// TwinCAT 3 PLC project plc_kfe_rix_vac
// Title: plc-kfe-rix-vac
// Company: SLAC
// ProjectVersion: 0.0.0
// ProgramVersion: 3.1.4023.0
// libraries:
//   LCLS General, * (SLAC)
//   LCLS Vacuum, * (SLAC - LCLS)
//   LCLSVacuumSerialDriverLib, * (SLAC)
//   PMPS, * (SLAC - LCLS)
//   Tc2_DataExchange, * (Beckhoff Automation GmbH)
//   Tc2_SerialCom, * (Beckhoff Automation GmbH)
//   Tc2_Standard, * (Beckhoff Automation GmbH)
//   Tc2_System, * (Beckhoff Automation GmbH)
//   Tc2_TcpIp, * (Beckhoff Automation GmbH)
//   Tc2_Utilities, * (Beckhoff Automation GmbH)
//   Tc3_Module, * (Beckhoff Automation GmbH)
// project tree:
//   / CheckBounds.TcPOU (not stored), CheckDivDInt.TcPOU (not stored), CheckDivLInt.TcPOU (not stored), CheckDivLReal.TcPOU (not stored), CheckDivReal.TcPOU (not stored), CheckLRangeSigned.TcPOU (not stored), CheckLRangeUnsigned.TcPOU (not stored), CheckPointer.TcPOU (not stored), CheckRangeSigned.TcPOU (not stored), CheckRangeUnsigned.TcPOU (not stored), FSTask.TcTTO (not stored), PlcTask.TcTTO (not stored), Serial_COM.TcTTO (not stored)
//   DUTs/ ST_EXT_ILK.TcDUT (not stored)
//   GVLs/ GVL_RIX_INTF.TcGVL (not stored), GVL_KFE_RIX_VAC.TcGVL, GVL_RIX_VAC_FSV_PMPS.TcGVL (not stored), GVL_RIX_VAC_FS_DEVICES.TcGVL (not stored), GVL_Serial_Com.TcGVL, GVL_Variables.TcGVL
//   POUs/ FB_PRO_ADS.TcPOU (not stored), MAIN.TcPOU (not stored), FB_EXT_ILK.TcPOU (not stored), PRG_COM.TcPOU, PRG_RIX_INTF.TcPOU (not stored), PRG_KFE_RIX_VAC.TcPOU, PRG_KFE_RIX_VAC_FS.TcPOU (not stored), PRG_Roughing.TcPOU (not stored)
// real-time tasks:
//   TASK PlcTask: cycle T#10ms, priority 20, ADS port 350
//   TASK FSTask: cycle T#1ms, priority 19, ADS port 352
//   TASK Serial_COM: cycle T#10ms, priority 25, ADS port 351
// I/O:
//   DEVICE Device 1 (EtherCAT)
//   DEVICE Device 5 (EtherCAT)
// variable links:
//   plc_kfe_rix_vac Instance <-> Device 1 (EtherCAT)/B950_100H1_WALL (EK1100)/Term 118 (EL2624)
//     PlcTask Outputs/GVL_KFE_RIX_VAC.fb_SL1K2_EXIT_GCC_1.q_xHV_DIS <-> Channel 1/Output
//   plc_kfe_rix_vac Instance <-> Device 1 (EtherCAT)/B950_100H1_WALL (EK1100)/Term 119 (EL3174)
//     PlcTask Inputs/GVL_KFE_RIX_VAC.fb_SL1K2_EXIT_GCC_1.i_iPRESS_R <-> AI Standard Channel 1/Value
//     PlcTask Inputs/GVL_KFE_RIX_VAC.fb_SL1K2_EXIT_GPI_1.i_iPRESS_R <-> AI Standard Channel 2/Value
//   plc_kfe_rix_vac Instance <-> Device 1 (EtherCAT)/B950_100H1_WALL (EK1100)/Term 120 (EL1004)
//     PlcTask Inputs/GVL_KFE_RIX_VAC.fb_SL1K2_EXIT_VGC_1.i_xClsLS <-> Channel 2/Input
//     PlcTask Inputs/GVL_KFE_RIX_VAC.fb_SL1K2_EXIT_VGC_1.i_xOpnLS <-> Channel 1/Input
//   plc_kfe_rix_vac Instance <-> Device 1 (EtherCAT)/B950_100H1_WALL (EK1100)/Term 121 (EL2004)
//     PlcTask Outputs/GVL_KFE_RIX_VAC.fb_SL1K2_EXIT_VGC_1.q_xOPN_DO <-> Channel 1/Output
//   plc_kfe_rix_vac Instance <-> Device 1 (EtherCAT)/B950_100H1_WALL (EK1100)/Term 123 (EL1124)
//     PlcTask Inputs/GVL_KFE_RIX_VAC.fb_SL1K2_EXIT_GCC_1.i_xDisc_Active <-> Channel 2/Input
//     PlcTask Inputs/GVL_KFE_RIX_VAC.fb_SL1K2_EXIT_GCC_1.i_xHV_ON <-> Channel 1/Input
//   plc_kfe_rix_vac Instance <-> Device 1 (EtherCAT)/Term 1 (EK1200)/PMPS_FFO (EL2202)
//     FSTask Outputs/GVL_RIX_VAC_FSV_PMPS.g_FastFaultOutput2.q_xFastFaultOut <-> Channel 2/Output
//     PlcTask Outputs/GVL_Variables.g_FastFaultOutput1.q_xFastFaultOut <-> Channel 1/Output
//   plc_kfe_rix_vac Instance <-> Device 1 (EtherCAT)/Term 1 (EK1200)/PMPS_PRE
//     PlcTask Inputs/MAIN.fbArbiterIO.i_stCurrentBP <-> IO Inputs/CurrentBP
//     PlcTask Inputs/MAIN.fbArbiterIO.xTxPDO_state <-> SYNC Inputs/TxPDO state
//     PlcTask Inputs/MAIN.fbArbiterIO.xTxPDO_toggle <-> SYNC Inputs/TxPDO toggle
//     PlcTask Outputs/MAIN.fbArbiterIO.q_stRequestedBP <-> IO Outputs/RequestedBP
//   plc_kfe_rix_vac Instance <-> Device 1 (EtherCAT)/Term 1 (EK1200)/Term 11 (EL2794)
//     PlcTask Outputs/GVL_KFE_RIX_VAC.fb_RIX_ILK.q_xILK_OK_DO <-> Channel 1/Output
//   plc_kfe_rix_vac Instance <-> Device 1 (EtherCAT)/Term 1 (EK1200)/Term 3 (EL2794)
//     PlcTask Outputs/GVL_KFE_RIX_VAC.fb_MR1K2_SWITCH_PIP_1.q_xHVEna_DO <-> Channel 3/Output
//     PlcTask Outputs/GVL_KFE_RIX_VAC.fb_PC1K1_ZOS_PIP_1.q_xHVEna_DO <-> Channel 2/Output
//     PlcTask Outputs/GVL_KFE_RIX_VAC.fb_TV1K1_PLEG_PIP_1.q_xHVEna_DO <-> Channel 4/Output
//   plc_kfe_rix_vac Instance <-> Device 1 (EtherCAT)/Term 1 (EK1200)/Term 32 (EK1122)/B940-008-K0S15-PNL-03 EK1100/Term 13 (EL2624)
//     PlcTask Outputs/GVL_KFE_RIX_VAC.fb_MR1K2_SWITCH_GCC_1.q_xHV_DIS <-> Channel 3/Output
//     PlcTask Outputs/GVL_KFE_RIX_VAC.fb_PC1K1_ZOS_GCC_1.q_xHV_DIS <-> Channel 1/Output
//     PlcTask Outputs/GVL_KFE_RIX_VAC.fb_TV1K1_PLEG_GCC_1.q_xHV_DIS <-> Channel 2/Output
//   plc_kfe_rix_vac Instance <-> Device 1 (EtherCAT)/Term 1 (EK1200)/Term 32 (EK1122)/B940-008-K0S15-PNL-03 EK1100/Term 14 (EL1004)
//     PlcTask Inputs/GVL_KFE_RIX_VAC.fb_MR1K2_SWITCH_VGC_1.i_xClsLS <-> Channel 2/Input
//     PlcTask Inputs/GVL_KFE_RIX_VAC.fb_MR1K2_SWITCH_VGC_2.i_xClsLS <-> Channel 4/Input
//     PlcTask Inputs/GVL_KFE_RIX_VAC.fb_MR1K2_SWITCH_VGC_1.i_xOpnLS <-> Channel 1/Input
//     PlcTask Inputs/GVL_KFE_RIX_VAC.fb_MR1K2_SWITCH_VGC_2.i_xOpnLS <-> Channel 3/Input
//   plc_kfe_rix_vac Instance <-> Device 1 (EtherCAT)/Term 1 (EK1200)/Term 32 (EK1122)/B940-008-K0S15-PNL-03 EK1100/Term 15 (EL2004)
//     PlcTask Outputs/GVL_KFE_RIX_VAC.fb_MR1K2_SWITCH_VGC_1.q_xOPN_DO <-> Channel 1/Output
//     PlcTask Outputs/GVL_KFE_RIX_VAC.fb_MR1K2_SWITCH_VGC_2.q_xOPN_DO <-> Channel 2/Output
//   plc_kfe_rix_vac Instance <-> Device 1 (EtherCAT)/Term 1 (EK1200)/Term 32 (EK1122)/B940-008-K0S15-PNL-03 EK1100/Term 16 (EL3174-0002)
//     PlcTask Inputs/GVL_KFE_RIX_VAC.fb_MR1K2_SWITCH_GCC_1.i_iPRESS_R <-> AI Standard Channel 2/Value
//     PlcTask Inputs/GVL_KFE_RIX_VAC.fb_PC1K1_ZOS_GCC_1.i_iPRESS_R <-> AI Standard Channel 1/Value
//     PlcTask Inputs/GVL_KFE_RIX_VAC.fb_PC1K1_ZOS_GPI_1.i_iPRESS_R <-> AI Standard Channel 4/Value
//     PlcTask Inputs/GVL_KFE_RIX_VAC.fb_TV1K1_PLEG_GCC_1.i_iPRESS_R <-> AI Standard Channel 3/Value
//   plc_kfe_rix_vac Instance <-> Device 1 (EtherCAT)/Term 1 (EK1200)/Term 32 (EK1122)/B940-008-K0S15-PNL-03 EK1100/Term 17 (EL3174-0002)
//     PlcTask Inputs/GVL_KFE_RIX_VAC.fb_MR1K2_SWITCH_GPI_1.i_iPRESS_R <-> AI Standard Channel 1/Value
//     PlcTask Inputs/GVL_KFE_RIX_VAC.fb_TV1K1_PLEG_GPI_1.i_iPRESS_R <-> AI Standard Channel 2/Value
//   plc_kfe_rix_vac Instance <-> Device 1 (EtherCAT)/Term 1 (EK1200)/Term 32 (EK1122)/B940-008-K0S15-PNL-03 EK1100/Term 19 (EL1124)
//     PlcTask Inputs/GVL_KFE_RIX_VAC.fb_MR1K2_SWITCH_GCC_1.i_xDisc_Active <-> Channel 4/Input
//     PlcTask Inputs/GVL_KFE_RIX_VAC.fb_MR1K2_SWITCH_GCC_1.i_xHV_ON <-> Channel 3/Input
//     PlcTask Inputs/GVL_KFE_RIX_VAC.fb_PC1K1_ZOS_GCC_1.i_xDisc_Active <-> Channel 2/Input
//     PlcTask Inputs/GVL_KFE_RIX_VAC.fb_PC1K1_ZOS_GCC_1.i_xHV_ON <-> Channel 1/Input
//   plc_kfe_rix_vac Instance <-> Device 1 (EtherCAT)/Term 1 (EK1200)/Term 32 (EK1122)/B940-008-K0S15-PNL-03 EK1100/Term 20 (EL1124)
//     PlcTask Inputs/GVL_KFE_RIX_VAC.fb_TV1K1_PLEG_GCC_1.i_xDisc_Active <-> Channel 2/Input
//     PlcTask Inputs/GVL_KFE_RIX_VAC.fb_TV1K1_PLEG_GCC_1.i_xHV_ON <-> Channel 1/Input
//   plc_kfe_rix_vac Instance <-> Device 1 (EtherCAT)/Term 1 (EK1200)/Term 32 (EK1122)/B940-008-K0S15-PNL-03 FS/Term 34 (EL2202)
//     FSTask Outputs/GVL_RIX_VAC_FS_DEVICES.fb_TV1K2_VFS_1.q_xClose_A <-> Channel 1/Output
//     FSTask Outputs/GVL_RIX_VAC_FS_DEVICES.fb_TV1K2_VFS_1.q_xClose_B <-> Channel 2/Output
//   plc_kfe_rix_vac Instance <-> Device 1 (EtherCAT)/Term 1 (EK1200)/Term 32 (EK1122)/B940-008-K0S15-PNL-03 FS/Term 35 (EL2202)
//     FSTask Outputs/GVL_RIX_VAC_FS_DEVICES.fb_TV1K2_VFS_1.q_xClose_C <-> Channel 1/Output
//     FSTask Outputs/GVL_RIX_VAC_FS_DEVICES.fb_TV1K2_VFS_1.q_xOPN_DO <-> Channel 2/Output
//   plc_kfe_rix_vac Instance <-> Device 1 (EtherCAT)/Term 1 (EK1200)/Term 32 (EK1122)/B940-008-K0S15-PNL-03 FS/Term 36 (EL1004)
//     FSTask Inputs/GVL_RIX_VAC_FS_DEVICES.fb_TV1K2_VFS_1.i_xClsLS <-> Channel 1/Input
//     FSTask Inputs/GVL_RIX_VAC_FS_DEVICES.fb_TV1K2_VFS_1.i_xOpnLS <-> Channel 2/Input
//   plc_kfe_rix_vac Instance <-> Device 1 (EtherCAT)/Term 1 (EK1200)/Term 4 (EL3064)
//     PlcTask Inputs/GVL_KFE_RIX_VAC.fb_MR1K2_SWITCH_PIP_1.i_iPRESS <-> AI Standard Channel 3/Value
//     PlcTask Inputs/GVL_KFE_RIX_VAC.fb_PC1K1_ZOS_PIP_1.i_iPRESS <-> AI Standard Channel 2/Value
//     PlcTask Inputs/GVL_KFE_RIX_VAC.fb_TV1K1_PLEG_PIP_1.i_iPRESS <-> AI Standard Channel 4/Value
//   plc_kfe_rix_vac Instance <-> Device 1 (EtherCAT)/Term 1 (EK1200)/Term 45 (EK1521-0010)/Term 47 (EK1501-0010)/B950_233_R02 (E2) (EL2794)
//     PlcTask Outputs/GVL_KFE_RIX_VAC.fb_MR2K2_FLAT_PIP_1.q_xHVEna_DO <-> Channel 2/GVL_KFE_RIX_VAC.fb_MR2K2_FLAT_PIP_1.q_xHVEna_DO
//     PlcTask Outputs/GVL_KFE_RIX_VAC.fb_MR3K2_KBH_PIP_1.q_xHVEna_DO <-> Channel 3/GVL_KFE_RIX_VAC.fb_MR3K2_KBH_PIP_1.q_xHVEna_DO
//     PlcTask Outputs/GVL_KFE_RIX_VAC.fb_MR4K2_KBV_PIP_1.q_xHVEna_DO <-> Channel 4/GVL_KFE_RIX_VAC.fb_MR4K2_KBV_PIP_1.q_xHVEna_DO
//     PlcTask Outputs/GVL_KFE_RIX_VAC.fb_ST1K2_PPS_PIP_1.q_xHVEna_DO <-> Channel 1/GVL_KFE_RIX_VAC.fb_ST1K2_PPS_PIP_1.q_xHVEna_DO
//   plc_kfe_rix_vac Instance <-> Device 1 (EtherCAT)/Term 1 (EK1200)/Term 45 (EK1521-0010)/Term 47 (EK1501-0010)/B950_233_R02 (E3) (EL3064)
//     PlcTask Inputs/GVL_KFE_RIX_VAC.fb_MR2K2_FLAT_PIP_1.i_iPRESS <-> AI Standard Channel 2/GVL_KFE_RIX_VAC.fb_MR2K2_FLAT_PIP_1.i_iPRESS
//     PlcTask Inputs/GVL_KFE_RIX_VAC.fb_MR3K2_KBH_PIP_1.i_iPRESS <-> AI Standard Channel 3/GVL_KFE_RIX_VAC.fb_MR3K2_KBH_PIP_1.i_iPRESS
//     PlcTask Inputs/GVL_KFE_RIX_VAC.fb_MR4K2_KBV_PIP_1.i_iPRESS <-> AI Standard Channel 4/GVL_KFE_RIX_VAC.fb_MR4K2_KBV_PIP_1.i_iPRESS
//     PlcTask Inputs/GVL_KFE_RIX_VAC.fb_ST1K2_PPS_PIP_1.i_iPRESS <-> AI Standard Channel 1/GVL_KFE_RIX_VAC.fb_ST1K2_PPS_PIP_1.i_iPRESS
//   plc_kfe_rix_vac Instance <-> Device 1 (EtherCAT)/Term 1 (EK1200)/Term 45 (EK1521-0010)/Term 47 (EK1501-0010)/B950_233_R02 (E4) (EL1004)
//     PlcTask Inputs/GVL_KFE_RIX_VAC.fb_MR2K2_FLAT_PIP_1.i_xSP_DI <-> Channel 2/GVL_KFE_RIX_VAC.fb_MR2K2_FLAT_PIP_1.i_xSP_DI
//     PlcTask Inputs/GVL_KFE_RIX_VAC.fb_MR3K2_KBH_PIP_1.i_xSP_DI <-> Channel 3/GVL_KFE_RIX_VAC.fb_MR3K2_KBH_PIP_1.i_xSP_DI
//     PlcTask Inputs/GVL_KFE_RIX_VAC.fb_MR4K2_KBV_PIP_1.i_xSP_DI <-> Channel 4/GVL_KFE_RIX_VAC.fb_MR4K2_KBV_PIP_1.i_xSP_DI
//     PlcTask Inputs/GVL_KFE_RIX_VAC.fb_ST1K2_PPS_PIP_1.i_xSP_DI <-> Channel 1/GVL_KFE_RIX_VAC.fb_ST1K2_PPS_PIP_1.i_xSP_DI
//   plc_kfe_rix_vac Instance <-> Device 1 (EtherCAT)/Term 1 (EK1200)/Term 45 (EK1521-0010)/Term 47 (EK1501-0010)/Term 52 (EL2794)
//     PlcTask Outputs/GVL_KFE_RIX_VAC.fb_IM5K2_PPM_PIP_1.q_xHVEna_DO <-> Channel 1/GVL_KFE_RIX_VAC.fb_IM5K2_PPM_PIP_1.q_xHVEna_DO
//     PlcTask Outputs/GVL_KFE_RIX_VAC.fb_SP1K2_PAX_PIP_1.q_xHVEna_DO <-> Channel 2/Output
//     PlcTask Outputs/GVL_KFE_RIX_VAC.fb_TV4K2_PIP_1.q_xHVEna_DO <-> Channel 4/GVL_KFE_RIX_VAC.fb_TV4K2_PIP_1.q_xHVEna_DO
//   plc_kfe_rix_vac Instance <-> Device 1 (EtherCAT)/Term 1 (EK1200)/Term 45 (EK1521-0010)/Term 47 (EK1501-0010)/Term 53 (EL3064)
//     PlcTask Inputs/GVL_KFE_RIX_VAC.fb_IM5K2_PPM_PIP_1.i_iPRESS <-> AI Standard Channel 1/GVL_KFE_RIX_VAC.fb_IM5K2_PPM_PIP_1.i_iPRESS
//     PlcTask Inputs/GVL_KFE_RIX_VAC.fb_SP1K2_PAX_PIP_1.i_iPRESS <-> AI Standard Channel 2/Value
//     PlcTask Inputs/GVL_KFE_RIX_VAC.fb_TV4K2_PIP_1.i_iPRESS <-> AI Standard Channel 4/GVL_KFE_RIX_VAC.fb_TV4K2_PIP_1.i_iPRESS
//   plc_kfe_rix_vac Instance <-> Device 1 (EtherCAT)/Term 1 (EK1200)/Term 45 (EK1521-0010)/Term 47 (EK1501-0010)/Term 54 (EL1004)
//     PlcTask Inputs/GVL_KFE_RIX_VAC.fb_IM5K2_PPM_PIP_1.i_xSP_DI <-> Channel 1/GVL_KFE_RIX_VAC.fb_IM5K2_PPM_PIP_1.i_xSP_DI
//     PlcTask Inputs/GVL_KFE_RIX_VAC.fb_SP1K2_PAX_PIP_1.i_xSP_DI <-> Channel 2/Input
//     PlcTask Inputs/GVL_KFE_RIX_VAC.fb_TV4K2_PIP_1.i_xSP_DI <-> Channel 4/GVL_KFE_RIX_VAC.fb_TV4K2_PIP_1.i_xSP_DI
//   plc_kfe_rix_vac Instance <-> Device 1 (EtherCAT)/Term 1 (EK1200)/Term 45 (EK1521-0010)/Term 47 (EK1501-0010)/Term 56 (EL2794)
//     PlcTask Outputs/GVL_KFE_RIX_VAC.fb_PA1K2_PIP_1.q_xHVEna_DO <-> Channel 1/GVL_KFE_RIX_VAC.fb_PA1K2_PIP_1.q_xHVEna_DO
//   plc_kfe_rix_vac Instance <-> Device 1 (EtherCAT)/Term 1 (EK1200)/Term 45 (EK1521-0010)/Term 47 (EK1501-0010)/Term 57 (EL3064)
//     PlcTask Inputs/GVL_KFE_RIX_VAC.fb_PA1K2_PIP_1.i_iPRESS <-> AI Standard Channel 1/GVL_KFE_RIX_VAC.fb_PA1K2_PIP_1.i_iPRESS
//   plc_kfe_rix_vac Instance <-> Device 1 (EtherCAT)/Term 1 (EK1200)/Term 45 (EK1521-0010)/Term 47 (EK1501-0010)/Term 58 (EL1004)
//     PlcTask Inputs/GVL_KFE_RIX_VAC.fb_PA1K2_PIP_1.i_xSP_DI <-> Channel 1/GVL_KFE_RIX_VAC.fb_PA1K2_PIP_1.i_xSP_DI
//   plc_kfe_rix_vac Instance <-> Device 1 (EtherCAT)/Term 1 (EK1200)/Term 45 (EK1521-0010)/Term 47 (EK1501-0010)/Term 59 (EL2794)
//     PlcTask Outputs/GVL_KFE_RIX_VAC.fb_IM2K2_PPM_PIP_1.q_xHVEna_DO <-> Channel 1/GVL_KFE_RIX_VAC.fb_IM2K2_PPM_PIP_1.q_xHVEna_DO
//     PlcTask Outputs/GVL_KFE_RIX_VAC.fb_IM3K2_PPM_PIP_1.q_xHVEna_DO <-> Channel 2/GVL_KFE_RIX_VAC.fb_IM3K2_PPM_PIP_1.q_xHVEna_DO
//     PlcTask Outputs/GVL_KFE_RIX_VAC.fb_IM4K2_PPM_PIP_1.q_xHVEna_DO <-> Channel 3/GVL_KFE_RIX_VAC.fb_IM4K2_PPM_PIP_1.q_xHVEna_DO
//     PlcTask Outputs/GVL_KFE_RIX_VAC.fb_LI2K2_K2A_PIP_1.q_xHVEna_DO <-> Channel 4/GVL_KFE_RIX_VAC.fb_LI2K2_K2A_PIP_1.q_xHVEna_DO
//   plc_kfe_rix_vac Instance <-> Device 1 (EtherCAT)/Term 1 (EK1200)/Term 45 (EK1521-0010)/Term 47 (EK1501-0010)/Term 62 (EK1122)/Box 110 (EP2338-0002)
//     PlcTask Inputs/GVL_KFE_RIX_VAC.fb_SP1K2_PAX_VGC_1.i_xClsLS <-> Channel 6/Input
//     PlcTask Inputs/GVL_KFE_RIX_VAC.fb_SP1K2_PAX_VGC_1.i_xOpnLS <-> Channel 5/Input
//     PlcTask Inputs/GVL_KFE_RIX_VAC.fb_ST1K2_PPS_VGC_1.i_xClsLS <-> Channel 2/Input
//     PlcTask Inputs/GVL_KFE_RIX_VAC.fb_ST1K2_PPS_VGC_1.i_xOpnLS <-> Channel 1/Input
//     PlcTask Outputs/GVL_KFE_RIX_VAC.fb_SP1K2_PAX_VGC_1.q_xOPN_DO <-> Channel 15/Output
//     PlcTask Outputs/GVL_KFE_RIX_VAC.fb_ST1K2_PPS_VGC_1.q_xOPN_DO <-> Channel 11/Output
//   plc_kfe_rix_vac Instance <-> Device 1 (EtherCAT)/Term 1 (EK1200)/Term 45 (EK1521-0010)/Term 47 (EK1501-0010)/Term 62 (EK1122)/Box 111 (EP3174-0002)
//     PlcTask Inputs/GVL_KFE_RIX_VAC.fb_ST1K2_PPS_GCC_1.i_iPRESS_R <-> AI Standard Channel 1/Value
//     PlcTask Inputs/GVL_KFE_RIX_VAC.fb_ST1K2_PPS_GPI_1.i_iPRESS_R <-> AI Standard Channel 2/Value
//   plc_kfe_rix_vac Instance <-> Device 1 (EtherCAT)/Term 1 (EK1200)/Term 45 (EK1521-0010)/Term 47 (EK1501-0010)/Term 62 (EK1122)/Box 256 (EP3174-0002)
//     PlcTask Inputs/GVL_KFE_RIX_VAC.fb_AT3K2_SOLID_GCP_1.i_iPRESS_R <-> AI Standard Channel 2/Value
//     PlcTask Inputs/GVL_KFE_RIX_VAC.fb_AT3K2_SOLID_GPI_1.i_iPRESS_R <-> AI Standard Channel 3/Value
//     PlcTask Inputs/GVL_KFE_RIX_VAC.fb_SP2K2_TXAS_GCP_1.i_iPRESS_R <-> AI Standard Channel 4/Value
//   plc_kfe_rix_vac Instance <-> Device 1 (EtherCAT)/Term 1 (EK1200)/Term 45 (EK1521-0010)/Term 47 (EK1501-0010)/Term 62 (EK1122)/EK1100_03_00/EL1004_03_01
//     PlcTask Inputs/GVL_KFE_RIX_VAC.fb_MR2K2_FLAT_VGC_1.i_xClsLS <-> Channel 2/GVL_KFE_RIX_VAC.fb_MR2K2_FLAT_VGC_1.i_xClsLS
//     PlcTask Inputs/GVL_KFE_RIX_VAC.fb_MR2K2_FLAT_VGC_2.i_xClsLS <-> Channel 4/GVL_KFE_RIX_VAC.fb_MR2K2_FLAT_VGC_2.i_xClsLS
//     PlcTask Inputs/GVL_KFE_RIX_VAC.fb_MR2K2_FLAT_VGC_1.i_xOpnLS <-> Channel 1/GVL_KFE_RIX_VAC.fb_MR2K2_FLAT_VGC_1.i_xOpnLS
//     PlcTask Inputs/GVL_KFE_RIX_VAC.fb_MR2K2_FLAT_VGC_2.i_xOpnLS <-> Channel 3/GVL_KFE_RIX_VAC.fb_MR2K2_FLAT_VGC_2.i_xOpnLS
//   plc_kfe_rix_vac Instance <-> Device 1 (EtherCAT)/Term 1 (EK1200)/Term 45 (EK1521-0010)/Term 47 (EK1501-0010)/Term 62 (EK1122)/EK1100_03_00/EL1004_03_03
//     PlcTask Inputs/GVL_KFE_RIX_VAC.fb_MR3K2_KBH_VGC_1.i_xClsLS <-> Channel 2/GVL_KFE_RIX_VAC.fb_MR3K2_KBH_VGC_1.i_xClsLS
//     PlcTask Inputs/GVL_KFE_RIX_VAC.fb_MR3K2_KBH_VGC_2.i_xClsLS <-> Channel 4/GVL_KFE_RIX_VAC.fb_MR3K2_KBH_VGC_2.i_xClsLS
//     PlcTask Inputs/GVL_KFE_RIX_VAC.fb_MR3K2_KBH_VGC_1.i_xOpnLS <-> Channel 1/GVL_KFE_RIX_VAC.fb_MR3K2_KBH_VGC_1.i_xOpnLS
//     PlcTask Inputs/GVL_KFE_RIX_VAC.fb_MR3K2_KBH_VGC_2.i_xOpnLS <-> Channel 3/GVL_KFE_RIX_VAC.fb_MR3K2_KBH_VGC_2.i_xOpnLS
//   plc_kfe_rix_vac Instance <-> Device 1 (EtherCAT)/Term 1 (EK1200)/Term 45 (EK1521-0010)/Term 47 (EK1501-0010)/Term 62 (EK1122)/EK1100_03_00/EL1124_03_10
//     PlcTask Inputs/GVL_KFE_RIX_VAC.fb_MR2K2_FLAT_GCC_1.i_xDisc_Active <-> Channel 2/GVL_KFE_RIX_VAC.fb_MR2K2_FLAT_GCC_1.i_xDisc_Active
//     PlcTask Inputs/GVL_KFE_RIX_VAC.fb_MR2K2_FLAT_GCC_1.i_xHV_ON <-> Channel 1/GVL_KFE_RIX_VAC.fb_MR2K2_FLAT_GCC_1.i_xHV_ON
//   plc_kfe_rix_vac Instance <-> Device 1 (EtherCAT)/Term 1 (EK1200)/Term 45 (EK1521-0010)/Term 47 (EK1501-0010)/Term 62 (EK1122)/EK1100_03_00/EL1124_03_11
//     PlcTask Inputs/GVL_KFE_RIX_VAC.fb_IM2K2_PPM_GCC_1.i_xDisc_Active <-> Channel 4/GVL_KFE_RIX_VAC.fb_IM2K2_PPM_GCC_1.i_xDisc_Active
//     PlcTask Inputs/GVL_KFE_RIX_VAC.fb_IM2K2_PPM_GCC_1.i_xHV_ON <-> Channel 3/GVL_KFE_RIX_VAC.fb_IM2K2_PPM_GCC_1.i_xHV_ON
//     PlcTask Inputs/GVL_KFE_RIX_VAC.fb_MR3K2_KBH_GCC_1.i_xDisc_Active <-> Channel 2/GVL_KFE_RIX_VAC.fb_MR3K2_KBH_GCC_1.i_xDisc_Active
//     PlcTask Inputs/GVL_KFE_RIX_VAC.fb_MR3K2_KBH_GCC_1.i_xHV_ON <-> Channel 1/GVL_KFE_RIX_VAC.fb_MR3K2_KBH_GCC_1.i_xHV_ON
//   plc_kfe_rix_vac Instance <-> Device 1 (EtherCAT)/Term 1 (EK1200)/Term 45 (EK1521-0010)/Term 47 (EK1501-0010)/Term 62 (EK1122)/EK1100_03_00/EL2004_03_02
//     PlcTask Outputs/GVL_KFE_RIX_VAC.fb_MR2K2_FLAT_VGC_1.q_xOPN_DO <-> Channel 1/GVL_KFE_RIX_VAC.fb_MR2K2_FLAT_VGC_1.q_xOPN_DO
//     PlcTask Outputs/GVL_KFE_RIX_VAC.fb_MR2K2_FLAT_VGC_2.q_xOPN_DO <-> Channel 2/GVL_KFE_RIX_VAC.fb_MR2K2_FLAT_VGC_2.q_xOPN_DO
//     PlcTask Outputs/GVL_KFE_RIX_VAC.fb_MR3K2_KBH_VGC_1.q_xOPN_DO <-> Channel 3/GVL_KFE_RIX_VAC.fb_MR3K2_KBH_VGC_1.q_xOPN_DO
//     PlcTask Outputs/GVL_KFE_RIX_VAC.fb_MR3K2_KBH_VGC_2.q_xOPN_DO <-> Channel 4/GVL_KFE_RIX_VAC.fb_MR3K2_KBH_VGC_2.q_xOPN_DO
//   plc_kfe_rix_vac Instance <-> Device 1 (EtherCAT)/Term 1 (EK1200)/Term 45 (EK1521-0010)/Term 47 (EK1501-0010)/Term 62 (EK1122)/EK1100_03_00/EL2624_03_08
//     PlcTask Outputs/GVL_KFE_RIX_VAC.fb_IM2K2_PPM_GCC_1.q_xHV_DIS <-> Channel 2/GVL_KFE_RIX_VAC.fb_IM2K2_PPM_GCC_1.q_xHV_DIS
//     PlcTask Outputs/GVL_KFE_RIX_VAC.fb_MR2K2_FLAT_GCC_1.q_xHV_DIS <-> Channel 1/GVL_KFE_RIX_VAC.fb_MR2K2_FLAT_GCC_1.q_xHV_DIS
//     PlcTask Outputs/GVL_KFE_RIX_VAC.fb_MR3K2_KBH_GCC_1.q_xHV_DIS <-> Channel 3/GVL_KFE_RIX_VAC.fb_MR3K2_KBH_GCC_1.q_xHV_DIS
//   plc_kfe_rix_vac Instance <-> Device 1 (EtherCAT)/Term 1 (EK1200)/Term 45 (EK1521-0010)/Term 47 (EK1501-0010)/Term 62 (EK1122)/EK1100_03_00/EL3174_03_12
//     PlcTask Inputs/GVL_KFE_RIX_VAC.fb_IM2K2_PPM_GCC_1.i_iPRESS_R <-> AI Standard Channel 2/GVL_KFE_RIX_VAC.fb_IM2K2_PPM_GCC_1.i_iPRESS_R
//     PlcTask Inputs/GVL_KFE_RIX_VAC.fb_MR2K2_FLAT_GCC_1.i_iPRESS_R <-> AI Standard Channel 1/GVL_KFE_RIX_VAC.fb_MR2K2_FLAT_GCC_1.i_iPRESS_R
//     PlcTask Inputs/GVL_KFE_RIX_VAC.fb_MR2K2_FLAT_GPI_1.i_iPRESS_R <-> AI Standard Channel 4/GVL_KFE_RIX_VAC.fb_MR2K2_FLAT_GPI_1.i_iPRESS_R
//     PlcTask Inputs/GVL_KFE_RIX_VAC.fb_MR3K2_KBH_GCC_1.i_iPRESS_R <-> AI Standard Channel 3/GVL_KFE_RIX_VAC.fb_MR3K2_KBH_GCC_1.i_iPRESS_R
//   plc_kfe_rix_vac Instance <-> Device 1 (EtherCAT)/Term 1 (EK1200)/Term 45 (EK1521-0010)/Term 47 (EK1501-0010)/Term 62 (EK1122)/EK1100_03_00/EL3174_03_13
//     PlcTask Inputs/GVL_KFE_RIX_VAC.fb_MR3K2_KBH_GPI_1.i_iPRESS_R <-> AI Standard Channel 1/GVL_KFE_RIX_VAC.fb_MR3K2_KBH_GPI_1.i_iPRESS_R
//   plc_kfe_rix_vac Instance <-> Device 1 (EtherCAT)/Term 1 (EK1200)/Term 45 (EK1521-0010)/Term 47 (EK1501-0010)/Term 62 (EK1122)/EK1100_04_00/EL1004_04_01
//     PlcTask Inputs/GVL_KFE_RIX_VAC.fb_MR4K2_KBV_VGC_1.i_xClsLS <-> Channel 2/GVL_KFE_RIX_VAC.fb_MR4K2_KBV_VGC_1.i_xClsLS
//     PlcTask Inputs/GVL_KFE_RIX_VAC.fb_MR4K2_KBV_VGC_2.i_xClsLS <-> Channel 4/GVL_KFE_RIX_VAC.fb_MR4K2_KBV_VGC_2.i_xClsLS
//     PlcTask Inputs/GVL_KFE_RIX_VAC.fb_MR4K2_KBV_VGC_1.i_xOpnLS <-> Channel 1/GVL_KFE_RIX_VAC.fb_MR4K2_KBV_VGC_1.i_xOpnLS
//     PlcTask Inputs/GVL_KFE_RIX_VAC.fb_MR4K2_KBV_VGC_2.i_xOpnLS <-> Channel 3/GVL_KFE_RIX_VAC.fb_MR4K2_KBV_VGC_2.i_xOpnLS
//   plc_kfe_rix_vac Instance <-> Device 1 (EtherCAT)/Term 1 (EK1200)/Term 45 (EK1521-0010)/Term 47 (EK1501-0010)/Term 62 (EK1122)/EK1100_04_00/EL1124_04_07
//     PlcTask Inputs/GVL_KFE_RIX_VAC.fb_IM3K2_PPM_GCC_1.i_xDisc_Active <-> Channel 2/GVL_KFE_RIX_VAC.fb_IM3K2_PPM_GCC_1.i_xDisc_Active
//     PlcTask Inputs/GVL_KFE_RIX_VAC.fb_IM3K2_PPM_GCC_1.i_xHV_ON <-> Channel 1/GVL_KFE_RIX_VAC.fb_IM3K2_PPM_GCC_1.i_xHV_ON
//     PlcTask Inputs/GVL_KFE_RIX_VAC.fb_MR4K2_KBV_GCC_1.i_xDisc_Active <-> Channel 4/GVL_KFE_RIX_VAC.fb_MR4K2_KBV_GCC_1.i_xDisc_Active
//     PlcTask Inputs/GVL_KFE_RIX_VAC.fb_MR4K2_KBV_GCC_1.i_xHV_ON <-> Channel 3/GVL_KFE_RIX_VAC.fb_MR4K2_KBV_GCC_1.i_xHV_ON
//   plc_kfe_rix_vac Instance <-> Device 1 (EtherCAT)/Term 1 (EK1200)/Term 45 (EK1521-0010)/Term 47 (EK1501-0010)/Term 62 (EK1122)/EK1100_04_00/EL1124_04_08
//     PlcTask Inputs/GVL_KFE_RIX_VAC.fb_IM4K2_PPM_GCC_1.i_xDisc_Active <-> Channel 2/GVL_KFE_RIX_VAC.fb_IM4K2_PPM_GCC_1.i_xDisc_Active
//     PlcTask Inputs/GVL_KFE_RIX_VAC.fb_IM4K2_PPM_GCC_1.i_xHV_ON <-> Channel 1/GVL_KFE_RIX_VAC.fb_IM4K2_PPM_GCC_1.i_xHV_ON
//   plc_kfe_rix_vac Instance <-> Device 1 (EtherCAT)/Term 1 (EK1200)/Term 45 (EK1521-0010)/Term 47 (EK1501-0010)/Term 62 (EK1122)/EK1100_04_00/EL2004_04_02
//     PlcTask Outputs/GVL_KFE_RIX_VAC.fb_MR4K2_KBV_VGC_1.q_xOPN_DO <-> Channel 1/GVL_KFE_RIX_VAC.fb_MR4K2_KBV_VGC_1.q_xOPN_DO
//     PlcTask Outputs/GVL_KFE_RIX_VAC.fb_MR4K2_KBV_VGC_2.q_xOPN_DO <-> Channel 2/GVL_KFE_RIX_VAC.fb_MR4K2_KBV_VGC_2.q_xOPN_DO
//   plc_kfe_rix_vac Instance <-> Device 1 (EtherCAT)/Term 1 (EK1200)/Term 45 (EK1521-0010)/Term 47 (EK1501-0010)/Term 62 (EK1122)/EK1100_04_00/EL2624_04_05
//     PlcTask Outputs/GVL_KFE_RIX_VAC.fb_IM3K2_PPM_GCC_1.q_xHV_DIS <-> Channel 1/GVL_KFE_RIX_VAC.fb_IM3K2_PPM_GCC_1.q_xHV_DIS
//     PlcTask Outputs/GVL_KFE_RIX_VAC.fb_IM4K2_PPM_GCC_1.q_xHV_DIS <-> Channel 3/GVL_KFE_RIX_VAC.fb_IM4K2_PPM_GCC_1.q_xHV_DIS
//     PlcTask Outputs/GVL_KFE_RIX_VAC.fb_MR4K2_KBV_GCC_1.q_xHV_DIS <-> Channel 2/GVL_KFE_RIX_VAC.fb_MR4K2_KBV_GCC_1.q_xHV_DIS
//   plc_kfe_rix_vac Instance <-> Device 1 (EtherCAT)/Term 1 (EK1200)/Term 45 (EK1521-0010)/Term 47 (EK1501-0010)/Term 62 (EK1122)/EK1100_04_00/EL3174_04_09
//     PlcTask Inputs/GVL_KFE_RIX_VAC.fb_IM3K2_PPM_GCC_1.i_iPRESS_R <-> AI Standard Channel 1/GVL_KFE_RIX_VAC.fb_IM3K2_PPM_GCC_1.i_iPRESS_R
//     PlcTask Inputs/GVL_KFE_RIX_VAC.fb_IM4K2_PPM_GCC_1.i_iPRESS_R <-> AI Standard Channel 3/GVL_KFE_RIX_VAC.fb_IM4K2_PPM_GCC_1.i_iPRESS_R
//     PlcTask Inputs/GVL_KFE_RIX_VAC.fb_MR4K2_KBV_GCC_1.i_iPRESS_R <-> AI Standard Channel 2/GVL_KFE_RIX_VAC.fb_MR4K2_KBV_GCC_1.i_iPRESS_R
//     PlcTask Inputs/GVL_KFE_RIX_VAC.fb_MR4K2_KBV_GPI_1.i_iPRESS_R <-> AI Standard Channel 4/GVL_KFE_RIX_VAC.fb_MR4K2_KBV_GPI_1.i_iPRESS_R
//   plc_kfe_rix_vac Instance <-> Device 1 (EtherCAT)/Term 1 (EK1200)/Term 45 (EK1521-0010)/Term 47 (EK1501-0010)/Term 62 (EK1122)/K2S13-DRL-01/EL1004_05_01
//     PlcTask Inputs/GVL_KFE_RIX_VAC.fb_LI2K2_K2A_VWC_1.i_xClsLS <-> Channel 4/Input
//     PlcTask Inputs/GVL_KFE_RIX_VAC.fb_LI2K2_K2A_VWC_1.i_xOpnLS <-> Channel 3/Input
//     PlcTask Inputs/GVL_KFE_RIX_VAC.fb_LI3K2_K2B_VWC_1.i_xClsLS <-> Channel 2/GVL_KFE_RIX_VAC.fb_LI3K2_K2B_VWC_1.i_xClsLS
//     PlcTask Inputs/GVL_KFE_RIX_VAC.fb_LI3K2_K2B_VWC_1.i_xOpnLS <-> Channel 1/GVL_KFE_RIX_VAC.fb_LI3K2_K2B_VWC_1.i_xOpnLS
//   plc_kfe_rix_vac Instance <-> Device 1 (EtherCAT)/Term 1 (EK1200)/Term 45 (EK1521-0010)/Term 47 (EK1501-0010)/Term 62 (EK1122)/K2S13-DRL-01/EL1004_05_03
//     PlcTask Inputs/GVL_KFE_RIX_VAC.fb_LI3K2_K2B_OUT_PTM_01.i_xAtSpd <-> Channel 1/Input
//     PlcTask Inputs/GVL_KFE_RIX_VAC.fb_LI3K2_K2B_OUT_PTM_01.i_xFaultNC <-> Channel 3/Input
//     PlcTask Inputs/GVL_KFE_RIX_VAC.fb_LI3K2_K2B_OUT_PTM_01.i_xRemote <-> Channel 2/Input
//   plc_kfe_rix_vac Instance <-> Device 1 (EtherCAT)/Term 1 (EK1200)/Term 45 (EK1521-0010)/Term 47 (EK1501-0010)/Term 62 (EK1122)/K2S13-DRL-01/EL1124_05_09
//     PlcTask Inputs/GVL_KFE_RIX_VAC.fb_IM5K2_PPM_GCC_1.i_xDisc_Active <-> Channel 4/GVL_KFE_RIX_VAC.fb_IM5K2_PPM_GCC_1.i_xDisc_Active
//     PlcTask Inputs/GVL_KFE_RIX_VAC.fb_IM5K2_PPM_GCC_1.i_xHV_ON <-> Channel 3/GVL_KFE_RIX_VAC.fb_IM5K2_PPM_GCC_1.i_xHV_ON
//   plc_kfe_rix_vac Instance <-> Device 1 (EtherCAT)/Term 1 (EK1200)/Term 45 (EK1521-0010)/Term 47 (EK1501-0010)/Term 62 (EK1122)/K2S13-DRL-01/EL1124_05_10
//     PlcTask Inputs/GVL_KFE_RIX_VAC.fb_TM2K2_K2B_GCC_1.i_xDisc_Active <-> Channel 2/GVL_KFE_RIX_VAC.fb_TM2K2_K2B_GCC_1.i_xDisc_Active
//     PlcTask Inputs/GVL_KFE_RIX_VAC.fb_TM2K2_K2B_GCC_1.i_xHV_ON <-> Channel 1/GVL_KFE_RIX_VAC.fb_TM2K2_K2B_GCC_1.i_xHV_ON
//   plc_kfe_rix_vac Instance <-> Device 1 (EtherCAT)/Term 1 (EK1200)/Term 45 (EK1521-0010)/Term 47 (EK1501-0010)/Term 62 (EK1122)/K2S13-DRL-01/EL2004_05_02
//     PlcTask Outputs/GVL_KFE_RIX_VAC.fb_LI2K2_K2A_VWC_1.q_xOPN_DO <-> Channel 2/Output
//     PlcTask Outputs/GVL_KFE_RIX_VAC.fb_LI3K2_K2B_VWC_1.q_xOPN_DO <-> Channel 1/GVL_KFE_RIX_VAC.fb_LI3K2_K2B_VWC_1.q_xOPN_DO
//   plc_kfe_rix_vac Instance <-> Device 1 (EtherCAT)/Term 1 (EK1200)/Term 45 (EK1521-0010)/Term 47 (EK1501-0010)/Term 62 (EK1122)/K2S13-DRL-01/EL2004_05_04
//     PlcTask Outputs/GVL_KFE_RIX_VAC.fb_LI3K2_K2B_OUT_PTM_01.q_PumpingStation <-> Channel 3/Output
//     PlcTask Outputs/GVL_KFE_RIX_VAC.fb_LI3K2_K2B_OUT_PTM_01.q_RunDO <-> Channel 1/Output
//     PlcTask Outputs/GVL_KFE_RIX_VAC.fb_LI3K2_K2B_OUT_PTM_01.q_xRemote <-> Channel 2/Output
//   plc_kfe_rix_vac Instance <-> Device 1 (EtherCAT)/Term 1 (EK1200)/Term 45 (EK1521-0010)/Term 47 (EK1501-0010)/Term 62 (EK1122)/K2S13-DRL-01/EL2624_05_07
//     PlcTask Outputs/GVL_KFE_RIX_VAC.fb_IM5K2_PPM_GCC_1.q_xHV_DIS <-> Channel 2/GVL_KFE_RIX_VAC.fb_IM5K2_PPM_GCC_1.q_xHV_DIS
//     PlcTask Outputs/GVL_KFE_RIX_VAC.fb_TM2K2_K2B_GCC_1.q_xHV_DIS <-> Channel 3/GVL_KFE_RIX_VAC.fb_TM2K2_K2B_GCC_1.q_xHV_DIS
//   plc_kfe_rix_vac Instance <-> Device 1 (EtherCAT)/Term 1 (EK1200)/Term 45 (EK1521-0010)/Term 47 (EK1501-0010)/Term 62 (EK1122)/K2S13-DRL-01/EL3174_05_11
//     PlcTask Inputs/GVL_KFE_RIX_VAC.fb_IM5K2_PPM_GCC_1.i_iPRESS_R <-> AI Standard Channel 2/GVL_KFE_RIX_VAC.fb_IM5K2_PPM_GCC_1.i_iPRESS_R
//     PlcTask Inputs/GVL_KFE_RIX_VAC.fb_IM5K2_PPM_GPI_1.i_iPRESS_R <-> AI Standard Channel 1/Value
//     PlcTask Inputs/GVL_KFE_RIX_VAC.fb_TM2K2_ATM_GPI_1.i_iPRESS_R <-> AI Standard Channel 4/GVL_KFE_RIX_VAC.fb_TM2K2_K2B_GPI_1.i_iPRESS_R
//     PlcTask Inputs/GVL_KFE_RIX_VAC.fb_TM2K2_K2B_GCC_1.i_iPRESS_R <-> AI Standard Channel 3/GVL_KFE_RIX_VAC.fb_TM2K2_K2B_GCC_1.i_iPRESS_R
//   plc_kfe_rix_vac Instance <-> Device 1 (EtherCAT)/Term 1 (EK1200)/Term 45 (EK1521-0010)/Term 47 (EK1501-0010)/Term 62 (EK1122)/K2S13-DRL-01/EL6021_05_12
//     Serial_COM Inputs/GVL_Serial_Com.stComIn_LI3K2_K2B_OUT_PTM_01/D[0] <-> COM TxPDO-Map Inputs/Data In 0
//     Serial_COM Inputs/GVL_Serial_Com.stComIn_LI3K2_K2B_OUT_PTM_01/D[10] <-> COM TxPDO-Map Inputs/Data In 10
//     Serial_COM Inputs/GVL_Serial_Com.stComIn_LI3K2_K2B_OUT_PTM_01/D[11] <-> COM TxPDO-Map Inputs/Data In 11
//     Serial_COM Inputs/GVL_Serial_Com.stComIn_LI3K2_K2B_OUT_PTM_01/D[12] <-> COM TxPDO-Map Inputs/Data In 12
//     Serial_COM Inputs/GVL_Serial_Com.stComIn_LI3K2_K2B_OUT_PTM_01/D[13] <-> COM TxPDO-Map Inputs/Data In 13
//     Serial_COM Inputs/GVL_Serial_Com.stComIn_LI3K2_K2B_OUT_PTM_01/D[14] <-> COM TxPDO-Map Inputs/Data In 14
//     Serial_COM Inputs/GVL_Serial_Com.stComIn_LI3K2_K2B_OUT_PTM_01/D[15] <-> COM TxPDO-Map Inputs/Data In 15
//     Serial_COM Inputs/GVL_Serial_Com.stComIn_LI3K2_K2B_OUT_PTM_01/D[16] <-> COM TxPDO-Map Inputs/Data In 16
//     Serial_COM Inputs/GVL_Serial_Com.stComIn_LI3K2_K2B_OUT_PTM_01/D[17] <-> COM TxPDO-Map Inputs/Data In 17
//     Serial_COM Inputs/GVL_Serial_Com.stComIn_LI3K2_K2B_OUT_PTM_01/D[18] <-> COM TxPDO-Map Inputs/Data In 18
//     Serial_COM Inputs/GVL_Serial_Com.stComIn_LI3K2_K2B_OUT_PTM_01/D[19] <-> COM TxPDO-Map Inputs/Data In 19
//     Serial_COM Inputs/GVL_Serial_Com.stComIn_LI3K2_K2B_OUT_PTM_01/D[1] <-> COM TxPDO-Map Inputs/Data In 1
//     Serial_COM Inputs/GVL_Serial_Com.stComIn_LI3K2_K2B_OUT_PTM_01/D[20] <-> COM TxPDO-Map Inputs/Data In 20
//     Serial_COM Inputs/GVL_Serial_Com.stComIn_LI3K2_K2B_OUT_PTM_01/D[21] <-> COM TxPDO-Map Inputs/Data In 21
//     Serial_COM Inputs/GVL_Serial_Com.stComIn_LI3K2_K2B_OUT_PTM_01/D[2] <-> COM TxPDO-Map Inputs/Data In 2
//     Serial_COM Inputs/GVL_Serial_Com.stComIn_LI3K2_K2B_OUT_PTM_01/D[3] <-> COM TxPDO-Map Inputs/Data In 3
//     Serial_COM Inputs/GVL_Serial_Com.stComIn_LI3K2_K2B_OUT_PTM_01/D[4] <-> COM TxPDO-Map Inputs/Data In 4
//     Serial_COM Inputs/GVL_Serial_Com.stComIn_LI3K2_K2B_OUT_PTM_01/D[5] <-> COM TxPDO-Map Inputs/Data In 5
//     Serial_COM Inputs/GVL_Serial_Com.stComIn_LI3K2_K2B_OUT_PTM_01/D[6] <-> COM TxPDO-Map Inputs/Data In 6
//     Serial_COM Inputs/GVL_Serial_Com.stComIn_LI3K2_K2B_OUT_PTM_01/D[7] <-> COM TxPDO-Map Inputs/Data In 7
//     Serial_COM Inputs/GVL_Serial_Com.stComIn_LI3K2_K2B_OUT_PTM_01/D[8] <-> COM TxPDO-Map Inputs/Data In 8
//     Serial_COM Inputs/GVL_Serial_Com.stComIn_LI3K2_K2B_OUT_PTM_01/D[9] <-> COM TxPDO-Map Inputs/Data In 9
//     Serial_COM Inputs/GVL_Serial_Com.stComIn_LI3K2_K2B_OUT_PTM_01/Status <-> COM TxPDO-Map Inputs/Status
//     Serial_COM Outputs/GVL_Serial_Com.stComOut_LI3K2_K2B_OUT_PTM_01/Ctrl <-> COM RxPDO-Map Outputs/Ctrl
//     Serial_COM Outputs/GVL_Serial_Com.stComOut_LI3K2_K2B_OUT_PTM_01/D[0] <-> COM RxPDO-Map Outputs/Data Out 0
//     Serial_COM Outputs/GVL_Serial_Com.stComOut_LI3K2_K2B_OUT_PTM_01/D[10] <-> COM RxPDO-Map Outputs/Data Out 10
//     Serial_COM Outputs/GVL_Serial_Com.stComOut_LI3K2_K2B_OUT_PTM_01/D[11] <-> COM RxPDO-Map Outputs/Data Out 11
//     Serial_COM Outputs/GVL_Serial_Com.stComOut_LI3K2_K2B_OUT_PTM_01/D[12] <-> COM RxPDO-Map Outputs/Data Out 12
//     Serial_COM Outputs/GVL_Serial_Com.stComOut_LI3K2_K2B_OUT_PTM_01/D[13] <-> COM RxPDO-Map Outputs/Data Out 13
//     Serial_COM Outputs/GVL_Serial_Com.stComOut_LI3K2_K2B_OUT_PTM_01/D[14] <-> COM RxPDO-Map Outputs/Data Out 14
//     Serial_COM Outputs/GVL_Serial_Com.stComOut_LI3K2_K2B_OUT_PTM_01/D[15] <-> COM RxPDO-Map Outputs/Data Out 15
//     Serial_COM Outputs/GVL_Serial_Com.stComOut_LI3K2_K2B_OUT_PTM_01/D[16] <-> COM RxPDO-Map Outputs/Data Out 16
//     Serial_COM Outputs/GVL_Serial_Com.stComOut_LI3K2_K2B_OUT_PTM_01/D[17] <-> COM RxPDO-Map Outputs/Data Out 17
//     Serial_COM Outputs/GVL_Serial_Com.stComOut_LI3K2_K2B_OUT_PTM_01/D[18] <-> COM RxPDO-Map Outputs/Data Out 18
//     Serial_COM Outputs/GVL_Serial_Com.stComOut_LI3K2_K2B_OUT_PTM_01/D[19] <-> COM RxPDO-Map Outputs/Data Out 19
//     Serial_COM Outputs/GVL_Serial_Com.stComOut_LI3K2_K2B_OUT_PTM_01/D[1] <-> COM RxPDO-Map Outputs/Data Out 1
//     Serial_COM Outputs/GVL_Serial_Com.stComOut_LI3K2_K2B_OUT_PTM_01/D[20] <-> COM RxPDO-Map Outputs/Data Out 20
//     Serial_COM Outputs/GVL_Serial_Com.stComOut_LI3K2_K2B_OUT_PTM_01/D[21] <-> COM RxPDO-Map Outputs/Data Out 21
//     Serial_COM Outputs/GVL_Serial_Com.stComOut_LI3K2_K2B_OUT_PTM_01/D[2] <-> COM RxPDO-Map Outputs/Data Out 2
//     Serial_COM Outputs/GVL_Serial_Com.stComOut_LI3K2_K2B_OUT_PTM_01/D[3] <-> COM RxPDO-Map Outputs/Data Out 3
//     Serial_COM Outputs/GVL_Serial_Com.stComOut_LI3K2_K2B_OUT_PTM_01/D[4] <-> COM RxPDO-Map Outputs/Data Out 4
//     Serial_COM Outputs/GVL_Serial_Com.stComOut_LI3K2_K2B_OUT_PTM_01/D[5] <-> COM RxPDO-Map Outputs/Data Out 5
//     Serial_COM Outputs/GVL_Serial_Com.stComOut_LI3K2_K2B_OUT_PTM_01/D[6] <-> COM RxPDO-Map Outputs/Data Out 6
//     Serial_COM Outputs/GVL_Serial_Com.stComOut_LI3K2_K2B_OUT_PTM_01/D[7] <-> COM RxPDO-Map Outputs/Data Out 7
//     Serial_COM Outputs/GVL_Serial_Com.stComOut_LI3K2_K2B_OUT_PTM_01/D[8] <-> COM RxPDO-Map Outputs/Data Out 8
//     Serial_COM Outputs/GVL_Serial_Com.stComOut_LI3K2_K2B_OUT_PTM_01/D[9] <-> COM RxPDO-Map Outputs/Data Out 9
//   plc_kfe_rix_vac Instance <-> Device 1 (EtherCAT)/Term 1 (EK1200)/Term 45 (EK1521-0010)/Term 47 (EK1501-0010)/Term 62 (EK1122)/K2S18 (EK1100)/K2S18 _EL1004_E4
//     PlcTask Inputs/GVL_KFE_RIX_VAC.fb_LI4K2_K2B_OUT_PTM_01.i_xAtSpd <-> Channel 1/Input
//     PlcTask Inputs/GVL_KFE_RIX_VAC.fb_LI4K2_K2B_OUT_PTM_01.i_xFaultNC <-> Channel 3/Input
//     PlcTask Inputs/GVL_KFE_RIX_VAC.fb_LI4K2_K2B_OUT_PTM_01.i_xRemote <-> Channel 2/Input
//   plc_kfe_rix_vac Instance <-> Device 1 (EtherCAT)/Term 1 (EK1200)/Term 45 (EK1521-0010)/Term 47 (EK1501-0010)/Term 62 (EK1122)/K2S18 (EK1100)/K2S18_EL1004_E1
//     PlcTask Inputs/GVL_KFE_RIX_VAC.fb_AT3K2_SOLID_VWC_01.i_xClsLS <-> Channel 2/Input
//     PlcTask Inputs/GVL_KFE_RIX_VAC.fb_AT3K2_SOLID_VWC_01.i_xOpnLS <-> Channel 1/Input
//   plc_kfe_rix_vac Instance <-> Device 1 (EtherCAT)/Term 1 (EK1200)/Term 45 (EK1521-0010)/Term 47 (EK1501-0010)/Term 62 (EK1122)/K2S18 (EK1100)/K2S18_EL1004_E7
//     PlcTask Inputs/GVL_KFE_RIX_VAC.fb_IM6K2_TXAS_PTM_01.i_xAtSpd <-> Channel 1/Input
//     PlcTask Inputs/GVL_KFE_RIX_VAC.fb_IM6K2_TXAS_PTM_01.i_xFaultNC <-> Channel 3/Input
//     PlcTask Inputs/GVL_KFE_RIX_VAC.fb_IM6K2_TXAS_PTM_01.i_xRemote <-> Channel 2/Input
//   plc_kfe_rix_vac Instance <-> Device 1 (EtherCAT)/Term 1 (EK1200)/Term 45 (EK1521-0010)/Term 47 (EK1501-0010)/Term 62 (EK1122)/K2S18 (EK1100)/K2S18_EL2004_E2
//     PlcTask Outputs/GVL_KFE_RIX_VAC.fb_AT3K2_SOLID_VWC_01.q_xCLS_DO <-> Channel 1/Output
//   plc_kfe_rix_vac Instance <-> Device 1 (EtherCAT)/Term 1 (EK1200)/Term 45 (EK1521-0010)/Term 47 (EK1501-0010)/Term 62 (EK1122)/K2S18 (EK1100)/K2S18_EL2004_E5
//     PlcTask Outputs/GVL_KFE_RIX_VAC.fb_LI4K2_K2B_OUT_PTM_01.q_PumpingStation <-> Channel 3/Output
//     PlcTask Outputs/GVL_KFE_RIX_VAC.fb_LI4K2_K2B_OUT_PTM_01.q_RunDO <-> Channel 1/Output
//     PlcTask Outputs/GVL_KFE_RIX_VAC.fb_LI4K2_K2B_OUT_PTM_01.q_xRemote <-> Channel 2/Output
//   plc_kfe_rix_vac Instance <-> Device 1 (EtherCAT)/Term 1 (EK1200)/Term 45 (EK1521-0010)/Term 47 (EK1501-0010)/Term 62 (EK1122)/K2S18 (EK1100)/K2S18_EL2004_E8
//     PlcTask Outputs/GVL_KFE_RIX_VAC.fb_IM6K2_TXAS_PTM_01.q_PumpingStation <-> Channel 3/Output
//     PlcTask Outputs/GVL_KFE_RIX_VAC.fb_IM6K2_TXAS_PTM_01.q_RunDO <-> Channel 1/Output
//     PlcTask Outputs/GVL_KFE_RIX_VAC.fb_IM6K2_TXAS_PTM_01.q_xRemote <-> Channel 2/Output
//   plc_kfe_rix_vac Instance <-> Device 1 (EtherCAT)/Term 1 (EK1200)/Term 45 (EK1521-0010)/Term 47 (EK1501-0010)/Term 62 (EK1122)/K2S18 (EK1100)/K2S18_EL6021_E6
//     Serial_COM Inputs/GVL_Serial_Com.stComIn_LI4K2_K2B_OUT_PTM_01/D[0] <-> COM TxPDO-Map Inputs/Data In 0
//     Serial_COM Inputs/GVL_Serial_Com.stComIn_LI4K2_K2B_OUT_PTM_01/D[10] <-> COM TxPDO-Map Inputs/Data In 10
//     Serial_COM Inputs/GVL_Serial_Com.stComIn_LI4K2_K2B_OUT_PTM_01/D[11] <-> COM TxPDO-Map Inputs/Data In 11
//     Serial_COM Inputs/GVL_Serial_Com.stComIn_LI4K2_K2B_OUT_PTM_01/D[12] <-> COM TxPDO-Map Inputs/Data In 12
//     Serial_COM Inputs/GVL_Serial_Com.stComIn_LI4K2_K2B_OUT_PTM_01/D[13] <-> COM TxPDO-Map Inputs/Data In 13
//     Serial_COM Inputs/GVL_Serial_Com.stComIn_LI4K2_K2B_OUT_PTM_01/D[14] <-> COM TxPDO-Map Inputs/Data In 14
//     Serial_COM Inputs/GVL_Serial_Com.stComIn_LI4K2_K2B_OUT_PTM_01/D[15] <-> COM TxPDO-Map Inputs/Data In 15
//     Serial_COM Inputs/GVL_Serial_Com.stComIn_LI4K2_K2B_OUT_PTM_01/D[16] <-> COM TxPDO-Map Inputs/Data In 16
//     Serial_COM Inputs/GVL_Serial_Com.stComIn_LI4K2_K2B_OUT_PTM_01/D[17] <-> COM TxPDO-Map Inputs/Data In 17
//     Serial_COM Inputs/GVL_Serial_Com.stComIn_LI4K2_K2B_OUT_PTM_01/D[18] <-> COM TxPDO-Map Inputs/Data In 18
//     Serial_COM Inputs/GVL_Serial_Com.stComIn_LI4K2_K2B_OUT_PTM_01/D[19] <-> COM TxPDO-Map Inputs/Data In 19
//     Serial_COM Inputs/GVL_Serial_Com.stComIn_LI4K2_K2B_OUT_PTM_01/D[1] <-> COM TxPDO-Map Inputs/Data In 1
//     Serial_COM Inputs/GVL_Serial_Com.stComIn_LI4K2_K2B_OUT_PTM_01/D[20] <-> COM TxPDO-Map Inputs/Data In 20
//     Serial_COM Inputs/GVL_Serial_Com.stComIn_LI4K2_K2B_OUT_PTM_01/D[21] <-> COM TxPDO-Map Inputs/Data In 21
//     Serial_COM Inputs/GVL_Serial_Com.stComIn_LI4K2_K2B_OUT_PTM_01/D[2] <-> COM TxPDO-Map Inputs/Data In 2
//     Serial_COM Inputs/GVL_Serial_Com.stComIn_LI4K2_K2B_OUT_PTM_01/D[3] <-> COM TxPDO-Map Inputs/Data In 3
//     Serial_COM Inputs/GVL_Serial_Com.stComIn_LI4K2_K2B_OUT_PTM_01/D[4] <-> COM TxPDO-Map Inputs/Data In 4
//     Serial_COM Inputs/GVL_Serial_Com.stComIn_LI4K2_K2B_OUT_PTM_01/D[5] <-> COM TxPDO-Map Inputs/Data In 5
//     Serial_COM Inputs/GVL_Serial_Com.stComIn_LI4K2_K2B_OUT_PTM_01/D[6] <-> COM TxPDO-Map Inputs/Data In 6
//     Serial_COM Inputs/GVL_Serial_Com.stComIn_LI4K2_K2B_OUT_PTM_01/D[7] <-> COM TxPDO-Map Inputs/Data In 7
//     Serial_COM Inputs/GVL_Serial_Com.stComIn_LI4K2_K2B_OUT_PTM_01/D[8] <-> COM TxPDO-Map Inputs/Data In 8
//     Serial_COM Inputs/GVL_Serial_Com.stComIn_LI4K2_K2B_OUT_PTM_01/D[9] <-> COM TxPDO-Map Inputs/Data In 9
//     Serial_COM Inputs/GVL_Serial_Com.stComIn_LI4K2_K2B_OUT_PTM_01/Status <-> COM TxPDO-Map Inputs/Status
//     Serial_COM Outputs/GVL_Serial_Com.stComOut_LI4K2_K2B_OUT_PTM_01/Ctrl <-> COM RxPDO-Map Outputs/Ctrl
//     Serial_COM Outputs/GVL_Serial_Com.stComOut_LI4K2_K2B_OUT_PTM_01/D[0] <-> COM RxPDO-Map Outputs/Data Out 0
//     Serial_COM Outputs/GVL_Serial_Com.stComOut_LI4K2_K2B_OUT_PTM_01/D[10] <-> COM RxPDO-Map Outputs/Data Out 10
//     Serial_COM Outputs/GVL_Serial_Com.stComOut_LI4K2_K2B_OUT_PTM_01/D[11] <-> COM RxPDO-Map Outputs/Data Out 11
//     Serial_COM Outputs/GVL_Serial_Com.stComOut_LI4K2_K2B_OUT_PTM_01/D[12] <-> COM RxPDO-Map Outputs/Data Out 12
//     Serial_COM Outputs/GVL_Serial_Com.stComOut_LI4K2_K2B_OUT_PTM_01/D[13] <-> COM RxPDO-Map Outputs/Data Out 13
//     Serial_COM Outputs/GVL_Serial_Com.stComOut_LI4K2_K2B_OUT_PTM_01/D[14] <-> COM RxPDO-Map Outputs/Data Out 14
//     Serial_COM Outputs/GVL_Serial_Com.stComOut_LI4K2_K2B_OUT_PTM_01/D[15] <-> COM RxPDO-Map Outputs/Data Out 15
//     Serial_COM Outputs/GVL_Serial_Com.stComOut_LI4K2_K2B_OUT_PTM_01/D[16] <-> COM RxPDO-Map Outputs/Data Out 16
//     Serial_COM Outputs/GVL_Serial_Com.stComOut_LI4K2_K2B_OUT_PTM_01/D[17] <-> COM RxPDO-Map Outputs/Data Out 17
//     Serial_COM Outputs/GVL_Serial_Com.stComOut_LI4K2_K2B_OUT_PTM_01/D[18] <-> COM RxPDO-Map Outputs/Data Out 18
//     Serial_COM Outputs/GVL_Serial_Com.stComOut_LI4K2_K2B_OUT_PTM_01/D[19] <-> COM RxPDO-Map Outputs/Data Out 19
//     Serial_COM Outputs/GVL_Serial_Com.stComOut_LI4K2_K2B_OUT_PTM_01/D[1] <-> COM RxPDO-Map Outputs/Data Out 1
//     Serial_COM Outputs/GVL_Serial_Com.stComOut_LI4K2_K2B_OUT_PTM_01/D[20] <-> COM RxPDO-Map Outputs/Data Out 20
//     Serial_COM Outputs/GVL_Serial_Com.stComOut_LI4K2_K2B_OUT_PTM_01/D[21] <-> COM RxPDO-Map Outputs/Data Out 21
//     Serial_COM Outputs/GVL_Serial_Com.stComOut_LI4K2_K2B_OUT_PTM_01/D[2] <-> COM RxPDO-Map Outputs/Data Out 2
//     Serial_COM Outputs/GVL_Serial_Com.stComOut_LI4K2_K2B_OUT_PTM_01/D[3] <-> COM RxPDO-Map Outputs/Data Out 3
//     Serial_COM Outputs/GVL_Serial_Com.stComOut_LI4K2_K2B_OUT_PTM_01/D[4] <-> COM RxPDO-Map Outputs/Data Out 4
//     Serial_COM Outputs/GVL_Serial_Com.stComOut_LI4K2_K2B_OUT_PTM_01/D[5] <-> COM RxPDO-Map Outputs/Data Out 5
//     Serial_COM Outputs/GVL_Serial_Com.stComOut_LI4K2_K2B_OUT_PTM_01/D[6] <-> COM RxPDO-Map Outputs/Data Out 6
//     Serial_COM Outputs/GVL_Serial_Com.stComOut_LI4K2_K2B_OUT_PTM_01/D[7] <-> COM RxPDO-Map Outputs/Data Out 7
//     Serial_COM Outputs/GVL_Serial_Com.stComOut_LI4K2_K2B_OUT_PTM_01/D[8] <-> COM RxPDO-Map Outputs/Data Out 8
//     Serial_COM Outputs/GVL_Serial_Com.stComOut_LI4K2_K2B_OUT_PTM_01/D[9] <-> COM RxPDO-Map Outputs/Data Out 9
//   plc_kfe_rix_vac Instance <-> Device 1 (EtherCAT)/Term 1 (EK1200)/Term 45 (EK1521-0010)/Term 47 (EK1501-0010)/Term 62 (EK1122)/K2S18 (EK1100)/K2S18_EL6021_E9
//     Serial_COM Inputs/GVL_Serial_Com.stComIn_IM6K2_TXAS_PTM_01/D[0] <-> COM TxPDO-Map Inputs/Data In 0
//     Serial_COM Inputs/GVL_Serial_Com.stComIn_IM6K2_TXAS_PTM_01/D[10] <-> COM TxPDO-Map Inputs/Data In 10
//     Serial_COM Inputs/GVL_Serial_Com.stComIn_IM6K2_TXAS_PTM_01/D[11] <-> COM TxPDO-Map Inputs/Data In 11
//     Serial_COM Inputs/GVL_Serial_Com.stComIn_IM6K2_TXAS_PTM_01/D[12] <-> COM TxPDO-Map Inputs/Data In 12
//     Serial_COM Inputs/GVL_Serial_Com.stComIn_IM6K2_TXAS_PTM_01/D[13] <-> COM TxPDO-Map Inputs/Data In 13
//     Serial_COM Inputs/GVL_Serial_Com.stComIn_IM6K2_TXAS_PTM_01/D[14] <-> COM TxPDO-Map Inputs/Data In 14
//     Serial_COM Inputs/GVL_Serial_Com.stComIn_IM6K2_TXAS_PTM_01/D[15] <-> COM TxPDO-Map Inputs/Data In 15
//     Serial_COM Inputs/GVL_Serial_Com.stComIn_IM6K2_TXAS_PTM_01/D[16] <-> COM TxPDO-Map Inputs/Data In 16
//     Serial_COM Inputs/GVL_Serial_Com.stComIn_IM6K2_TXAS_PTM_01/D[17] <-> COM TxPDO-Map Inputs/Data In 17
//     Serial_COM Inputs/GVL_Serial_Com.stComIn_IM6K2_TXAS_PTM_01/D[18] <-> COM TxPDO-Map Inputs/Data In 18
//     Serial_COM Inputs/GVL_Serial_Com.stComIn_IM6K2_TXAS_PTM_01/D[19] <-> COM TxPDO-Map Inputs/Data In 19
//     Serial_COM Inputs/GVL_Serial_Com.stComIn_IM6K2_TXAS_PTM_01/D[1] <-> COM TxPDO-Map Inputs/Data In 1
//     Serial_COM Inputs/GVL_Serial_Com.stComIn_IM6K2_TXAS_PTM_01/D[20] <-> COM TxPDO-Map Inputs/Data In 20
//     Serial_COM Inputs/GVL_Serial_Com.stComIn_IM6K2_TXAS_PTM_01/D[21] <-> COM TxPDO-Map Inputs/Data In 21
//     Serial_COM Inputs/GVL_Serial_Com.stComIn_IM6K2_TXAS_PTM_01/D[2] <-> COM TxPDO-Map Inputs/Data In 2
//     Serial_COM Inputs/GVL_Serial_Com.stComIn_IM6K2_TXAS_PTM_01/D[3] <-> COM TxPDO-Map Inputs/Data In 3
//     Serial_COM Inputs/GVL_Serial_Com.stComIn_IM6K2_TXAS_PTM_01/D[4] <-> COM TxPDO-Map Inputs/Data In 4
//     Serial_COM Inputs/GVL_Serial_Com.stComIn_IM6K2_TXAS_PTM_01/D[5] <-> COM TxPDO-Map Inputs/Data In 5
//     Serial_COM Inputs/GVL_Serial_Com.stComIn_IM6K2_TXAS_PTM_01/D[6] <-> COM TxPDO-Map Inputs/Data In 6
//     Serial_COM Inputs/GVL_Serial_Com.stComIn_IM6K2_TXAS_PTM_01/D[7] <-> COM TxPDO-Map Inputs/Data In 7
//     Serial_COM Inputs/GVL_Serial_Com.stComIn_IM6K2_TXAS_PTM_01/D[8] <-> COM TxPDO-Map Inputs/Data In 8
//     Serial_COM Inputs/GVL_Serial_Com.stComIn_IM6K2_TXAS_PTM_01/D[9] <-> COM TxPDO-Map Inputs/Data In 9
//     Serial_COM Inputs/GVL_Serial_Com.stComIn_IM6K2_TXAS_PTM_01/Status <-> COM TxPDO-Map Inputs/Status
//     Serial_COM Outputs/GVL_Serial_Com.stComOut_IM6K2_TXAS_PTM_01/Ctrl <-> COM RxPDO-Map Outputs/Ctrl
//     Serial_COM Outputs/GVL_Serial_Com.stComOut_IM6K2_TXAS_PTM_01/D[0] <-> COM RxPDO-Map Outputs/Data Out 0
//     Serial_COM Outputs/GVL_Serial_Com.stComOut_IM6K2_TXAS_PTM_01/D[10] <-> COM RxPDO-Map Outputs/Data Out 10
//     Serial_COM Outputs/GVL_Serial_Com.stComOut_IM6K2_TXAS_PTM_01/D[11] <-> COM RxPDO-Map Outputs/Data Out 11
//     Serial_COM Outputs/GVL_Serial_Com.stComOut_IM6K2_TXAS_PTM_01/D[12] <-> COM RxPDO-Map Outputs/Data Out 12
//     Serial_COM Outputs/GVL_Serial_Com.stComOut_IM6K2_TXAS_PTM_01/D[13] <-> COM RxPDO-Map Outputs/Data Out 13
//     Serial_COM Outputs/GVL_Serial_Com.stComOut_IM6K2_TXAS_PTM_01/D[14] <-> COM RxPDO-Map Outputs/Data Out 14
//     Serial_COM Outputs/GVL_Serial_Com.stComOut_IM6K2_TXAS_PTM_01/D[15] <-> COM RxPDO-Map Outputs/Data Out 15
//     Serial_COM Outputs/GVL_Serial_Com.stComOut_IM6K2_TXAS_PTM_01/D[16] <-> COM RxPDO-Map Outputs/Data Out 16
//     Serial_COM Outputs/GVL_Serial_Com.stComOut_IM6K2_TXAS_PTM_01/D[17] <-> COM RxPDO-Map Outputs/Data Out 17
//     Serial_COM Outputs/GVL_Serial_Com.stComOut_IM6K2_TXAS_PTM_01/D[18] <-> COM RxPDO-Map Outputs/Data Out 18
//     Serial_COM Outputs/GVL_Serial_Com.stComOut_IM6K2_TXAS_PTM_01/D[19] <-> COM RxPDO-Map Outputs/Data Out 19
//     Serial_COM Outputs/GVL_Serial_Com.stComOut_IM6K2_TXAS_PTM_01/D[1] <-> COM RxPDO-Map Outputs/Data Out 1
//     Serial_COM Outputs/GVL_Serial_Com.stComOut_IM6K2_TXAS_PTM_01/D[20] <-> COM RxPDO-Map Outputs/Data Out 20
//     Serial_COM Outputs/GVL_Serial_Com.stComOut_IM6K2_TXAS_PTM_01/D[21] <-> COM RxPDO-Map Outputs/Data Out 21
//     Serial_COM Outputs/GVL_Serial_Com.stComOut_IM6K2_TXAS_PTM_01/D[2] <-> COM RxPDO-Map Outputs/Data Out 2
//     Serial_COM Outputs/GVL_Serial_Com.stComOut_IM6K2_TXAS_PTM_01/D[3] <-> COM RxPDO-Map Outputs/Data Out 3
//     Serial_COM Outputs/GVL_Serial_Com.stComOut_IM6K2_TXAS_PTM_01/D[4] <-> COM RxPDO-Map Outputs/Data Out 4
//     Serial_COM Outputs/GVL_Serial_Com.stComOut_IM6K2_TXAS_PTM_01/D[5] <-> COM RxPDO-Map Outputs/Data Out 5
//     Serial_COM Outputs/GVL_Serial_Com.stComOut_IM6K2_TXAS_PTM_01/D[6] <-> COM RxPDO-Map Outputs/Data Out 6
//     Serial_COM Outputs/GVL_Serial_Com.stComOut_IM6K2_TXAS_PTM_01/D[7] <-> COM RxPDO-Map Outputs/Data Out 7
//     Serial_COM Outputs/GVL_Serial_Com.stComOut_IM6K2_TXAS_PTM_01/D[8] <-> COM RxPDO-Map Outputs/Data Out 8
//     Serial_COM Outputs/GVL_Serial_Com.stComOut_IM6K2_TXAS_PTM_01/D[9] <-> COM RxPDO-Map Outputs/Data Out 9
//   plc_kfe_rix_vac Instance <-> Device 1 (EtherCAT)/Term 1 (EK1200)/Term 45 (EK1521-0010)/Term 47 (EK1501-0010)/Term 62 (EK1122)/K2S2-DRL-01 (EP2624-0002)
//     PlcTask Outputs/GVL_KFE_RIX_VAC.fb_ST1K2_PPS_GCC_1.q_xHV_DIS <-> Channel 1/Output
//   plc_kfe_rix_vac Instance <-> Device 1 (EtherCAT)/Term 1 (EK1200)/Term 45 (EK1521-0010)/Term 47 (EK1501-0010)/Term 62 (EK1122)/Term 63 (EK1100) B950-233-100H1-R02-DRL-02/Term 104 (EL2008)
//     PlcTask Outputs/PRG_RIX_INTF.FB_FIM_ILK <-> Channel 1/PRG_RIX_INTF.FB_FIM_ILK
//   plc_kfe_rix_vac Instance <-> Device 1 (EtherCAT)/Term 1 (EK1200)/Term 45 (EK1521-0010)/Term 47 (EK1501-0010)/Term 62 (EK1122)/Term 63 (EK1100) B950-233-100H1-R02-DRL-02/Term 164 (EL3174-0002)
//     PlcTask Inputs/GVL_KFE_RIX_VAC.fb_SP2K2_TXAS_PIP_1.i_iPRESS <-> AI Standard Channel 4/GVL_KFE_RIX_VAC.fb_SP2K2_TXAS_PIP_1.i_iPRESS
//   plc_kfe_rix_vac Instance <-> Device 1 (EtherCAT)/Term 1 (EK1200)/Term 45 (EK1521-0010)/Term 47 (EK1501-0010)/Term 62 (EK1122)/Term 63 (EK1100) B950-233-100H1-R02-DRL-02/Term 68 (EL3064)
//     PlcTask Inputs/GVL_KFE_RIX_VAC.fb_TV4K2_GFS_1.i_iPRESS_R <-> AI Standard Channel 1/Value
//   plc_kfe_rix_vac Instance <-> Device 1 (EtherCAT)/Term 1 (EK1200)/Term 45 (EK1521-0010)/Term 47 (EK1501-0010)/Term 62 (EK1122)/Term 63 (EK1100) B950-233-100H1-R02-DRL-02/Term 70 (EL2794)
//     PlcTask Outputs/GVL_KFE_RIX_VAC.fb_SP2K2_TXAS_PIP_1.q_xHVEna_DO <-> Channel 4/GVL_KFE_RIX_VAC.fb_SP2K2_TXAS_PIP_1.q_xHVEna_DO
//     PlcTask Outputs/GVL_KFE_RIX_VAC.fb_TV4K2_GFS_1.q_xHV_DIS <-> Channel 1/Output
//   plc_kfe_rix_vac Instance <-> Device 1 (EtherCAT)/Term 1 (EK1200)/Term 45 (EK1521-0010)/Term 47 (EK1501-0010)/Term 62 (EK1122)/Term 63 (EK1100) B950-233-100H1-R02-DRL-02/Term 72 (EL1124)
//     FSTask Inputs/GVL_RIX_VAC_FS_DEVICES.fb_TV1K2_VFS_1.i_xTrigger <-> Channel 1/GVL_RIX_VAC_FS_DEVICES.fb_TV1K2_VFS_1.i_xTrigger
//     PlcTask Inputs/GVL_KFE_RIX_VAC.fb_SP2K2_TXAS_PIP_1.i_xIP_ON <-> Channel 3/GVL_KFE_RIX_VAC.fb_SP2K2_TXAS_PIP_1.i_xIP_ON
//   plc_kfe_rix_vac Instance <-> Device 1 (EtherCAT)/Term 1 (EK1200)/Term 45 (EK1521-0010)/Term 47 (EK1501-0010)/Term 62 (EK1122)/Term 63 (EK1100) B950-233-100H1-R02-DRL-02/Term 77 (EK1122)/Term 201 (EK1100)/EL1088_03_01
//     PlcTask Inputs/GVL_KFE_RIX_VAC.RIXS_PRO_01.i_xAlarmOK <-> Channel 4/Input
//     PlcTask Inputs/GVL_KFE_RIX_VAC.RIXS_PRO_01.i_xBPStatus <-> Channel 2/Input
//     PlcTask Inputs/GVL_KFE_RIX_VAC.RIXS_PRO_01.i_xMPStatus <-> Channel 1/Input
//     PlcTask Inputs/GVL_KFE_RIX_VAC.RIXS_PRO_01.i_xWarning <-> Channel 3/Input
//   plc_kfe_rix_vac Instance <-> Device 1 (EtherCAT)/Term 1 (EK1200)/Term 45 (EK1521-0010)/Term 47 (EK1501-0010)/Term 62 (EK1122)/Term 63 (EK1100) B950-233-100H1-R02-DRL-02/Term 77 (EK1122)/Term 201 (EK1100)/EL2212_03_04
//     PlcTask Outputs/GVL_KFE_RIX_VAC.RIXS_ROUGH_VRO_01.q_xOPN_DO <-> DOX Control Channel 1/Control/Output
//   plc_kfe_rix_vac Instance <-> Device 1 (EtherCAT)/Term 1 (EK1200)/Term 45 (EK1521-0010)/Term 47 (EK1501-0010)/Term 62 (EK1122)/Term 63 (EK1100) B950-233-100H1-R02-DRL-02/Term 77 (EK1122)/Term 201 (EK1100)/EL2794_03_03
//     PlcTask Outputs/GVL_KFE_RIX_VAC.RIXS_PRO_01.q_xBPStart <-> Channel 2/Output
//     PlcTask Outputs/GVL_KFE_RIX_VAC.RIXS_PRO_01.q_xMPStart <-> Channel 1/Output
//   plc_kfe_rix_vac Instance <-> Device 1 (EtherCAT)/Term 1 (EK1200)/Term 45 (EK1521-0010)/Term 47 (EK1501-0010)/Term 62 (EK1122)/Term 63 (EK1100) B950-233-100H1-R02-DRL-02/Term 77 (EK1122)/Term 201 (EK1100)/EL3174-0002_03_07
//     PlcTask Inputs/GVL_KFE_RIX_VAC.RIXS_ROUGH_GPI_01.i_iPRESS_R <-> AI Standard Channel 4/Value
//   plc_kfe_rix_vac Instance <-> Device 1 (EtherCAT)/Term 1 (EK1200)/Term 45 (EK1521-0010)/Term 47 (EK1501-0010)/Term 62 (EK1122)/Term 63 (EK1100) B950-233-100H1-R02-DRL-02/Term 98 (EK1122)/Term 156 (EK1100) B950-233-PAX-DRL-01/Term 157 (EL1004)
//     PlcTask Inputs/GVL_KFE_RIX_VAC.fb_SP1K2_PAX_VRC_1.i_xClsLS <-> Channel 2/Input
//     PlcTask Inputs/GVL_KFE_RIX_VAC.fb_SP1K2_PAX_VRC_2.i_xClsLS <-> Channel 4/Input
//     PlcTask Inputs/GVL_KFE_RIX_VAC.fb_SP1K2_PAX_VRC_1.i_xOpnLS <-> Channel 1/Input
//     PlcTask Inputs/GVL_KFE_RIX_VAC.fb_SP1K2_PAX_VRC_2.i_xOpnLS <-> Channel 3/Input
//   plc_kfe_rix_vac Instance <-> Device 1 (EtherCAT)/Term 1 (EK1200)/Term 45 (EK1521-0010)/Term 47 (EK1501-0010)/Term 62 (EK1122)/Term 63 (EK1100) B950-233-100H1-R02-DRL-02/Term 98 (EK1122)/Term 156 (EK1100) B950-233-PAX-DRL-01/Term 158 (EL2004)
//     PlcTask Outputs/GVL_KFE_RIX_VAC.fb_SP1K2_PAX_VRC_1.q_xOPN_DO <-> Channel 1/Output
//     PlcTask Outputs/GVL_KFE_RIX_VAC.fb_SP1K2_PAX_VRC_2.q_xOPN_DO <-> Channel 2/Output
//     PlcTask Outputs/GVL_KFE_RIX_VAC.fb_SP1K2_PAX_VRM_3.q_xOPN_DO <-> Channel 3/Output
//   plc_kfe_rix_vac Instance <-> Device 1 (EtherCAT)/Term 1 (EK1200)/Term 45 (EK1521-0010)/Term 47 (EK1501-0010)/Term 62 (EK1122)/Term 63 (EK1100) B950-233-100H1-R02-DRL-02/Term 98 (EK1122)/Term 156 (EK1100) B950-233-PAX-DRL-01/Term 159 (EL1004)
//     PlcTask Inputs/GVL_KFE_RIX_VAC.fb_SP1K2_PAX_VRM_3.i_xClsLS <-> Channel 2/Input
//     PlcTask Inputs/GVL_KFE_RIX_VAC.fb_SP1K2_PAX_VRM_3.i_xOpnLS <-> Channel 1/Input
//   plc_kfe_rix_vac Instance <-> Device 1 (EtherCAT)/Term 1 (EK1200)/Term 45 (EK1521-0010)/Term 47 (EK1501-0010)/Term 62 (EK1122)/Term 63 (EK1100) B950-233-100H1-R02-DRL-02/Term 98 (EK1122)/Term 156 (EK1100) B950-233-PAX-DRL-01/Term 160 (EL1004)
//     PlcTask Inputs/GVL_KFE_RIX_VAC.fb_SP1K2_PAX_PTM_01.i_xAtSpd <-> Channel 1/Input
//     PlcTask Inputs/GVL_KFE_RIX_VAC.fb_SP1K2_PAX_PTM_01.i_xFaultNC <-> Channel 3/Input
//     PlcTask Inputs/GVL_KFE_RIX_VAC.fb_SP1K2_PAX_PTM_01.i_xRemote <-> Channel 2/Input
//   plc_kfe_rix_vac Instance <-> Device 1 (EtherCAT)/Term 1 (EK1200)/Term 45 (EK1521-0010)/Term 47 (EK1501-0010)/Term 62 (EK1122)/Term 63 (EK1100) B950-233-100H1-R02-DRL-02/Term 98 (EK1122)/Term 156 (EK1100) B950-233-PAX-DRL-01/Term 161 (EL2004)
//     PlcTask Outputs/GVL_KFE_RIX_VAC.fb_SP1K2_PAX_PTM_01.q_PumpingStation <-> Channel 3/Output
//     PlcTask Outputs/GVL_KFE_RIX_VAC.fb_SP1K2_PAX_PTM_01.q_RunDO <-> Channel 1/Output
//     PlcTask Outputs/GVL_KFE_RIX_VAC.fb_SP1K2_PAX_PTM_01.q_xRemote <-> Channel 2/Output
//   plc_kfe_rix_vac Instance <-> Device 1 (EtherCAT)/Term 1 (EK1200)/Term 45 (EK1521-0010)/Term 47 (EK1501-0010)/Term 62 (EK1122)/Term 63 (EK1100) B950-233-100H1-R02-DRL-02/Term 98 (EK1122)/Term 156 (EK1100) B950-233-PAX-DRL-01/Term 162 (EL6021)
//     Serial_COM Inputs/GVL_Serial_Com.stComIn_SP1K2_PAX_PTM_01/D[0] <-> COM TxPDO-Map Inputs/Data In 0
//     Serial_COM Inputs/GVL_Serial_Com.stComIn_SP1K2_PAX_PTM_01/D[10] <-> COM TxPDO-Map Inputs/Data In 10
//     Serial_COM Inputs/GVL_Serial_Com.stComIn_SP1K2_PAX_PTM_01/D[11] <-> COM TxPDO-Map Inputs/Data In 11
//     Serial_COM Inputs/GVL_Serial_Com.stComIn_SP1K2_PAX_PTM_01/D[12] <-> COM TxPDO-Map Inputs/Data In 12
//     Serial_COM Inputs/GVL_Serial_Com.stComIn_SP1K2_PAX_PTM_01/D[13] <-> COM TxPDO-Map Inputs/Data In 13
//     Serial_COM Inputs/GVL_Serial_Com.stComIn_SP1K2_PAX_PTM_01/D[14] <-> COM TxPDO-Map Inputs/Data In 14
//     Serial_COM Inputs/GVL_Serial_Com.stComIn_SP1K2_PAX_PTM_01/D[15] <-> COM TxPDO-Map Inputs/Data In 15
//     Serial_COM Inputs/GVL_Serial_Com.stComIn_SP1K2_PAX_PTM_01/D[16] <-> COM TxPDO-Map Inputs/Data In 16
//     Serial_COM Inputs/GVL_Serial_Com.stComIn_SP1K2_PAX_PTM_01/D[17] <-> COM TxPDO-Map Inputs/Data In 17
//     Serial_COM Inputs/GVL_Serial_Com.stComIn_SP1K2_PAX_PTM_01/D[18] <-> COM TxPDO-Map Inputs/Data In 18
//     Serial_COM Inputs/GVL_Serial_Com.stComIn_SP1K2_PAX_PTM_01/D[19] <-> COM TxPDO-Map Inputs/Data In 19
//     Serial_COM Inputs/GVL_Serial_Com.stComIn_SP1K2_PAX_PTM_01/D[1] <-> COM TxPDO-Map Inputs/Data In 1
//     Serial_COM Inputs/GVL_Serial_Com.stComIn_SP1K2_PAX_PTM_01/D[20] <-> COM TxPDO-Map Inputs/Data In 20
//     Serial_COM Inputs/GVL_Serial_Com.stComIn_SP1K2_PAX_PTM_01/D[21] <-> COM TxPDO-Map Inputs/Data In 21
//     Serial_COM Inputs/GVL_Serial_Com.stComIn_SP1K2_PAX_PTM_01/D[2] <-> COM TxPDO-Map Inputs/Data In 2
//     Serial_COM Inputs/GVL_Serial_Com.stComIn_SP1K2_PAX_PTM_01/D[3] <-> COM TxPDO-Map Inputs/Data In 3
//     Serial_COM Inputs/GVL_Serial_Com.stComIn_SP1K2_PAX_PTM_01/D[4] <-> COM TxPDO-Map Inputs/Data In 4
//     Serial_COM Inputs/GVL_Serial_Com.stComIn_SP1K2_PAX_PTM_01/D[5] <-> COM TxPDO-Map Inputs/Data In 5
//     Serial_COM Inputs/GVL_Serial_Com.stComIn_SP1K2_PAX_PTM_01/D[6] <-> COM TxPDO-Map Inputs/Data In 6
//     Serial_COM Inputs/GVL_Serial_Com.stComIn_SP1K2_PAX_PTM_01/D[7] <-> COM TxPDO-Map Inputs/Data In 7
//     Serial_COM Inputs/GVL_Serial_Com.stComIn_SP1K2_PAX_PTM_01/D[8] <-> COM TxPDO-Map Inputs/Data In 8
//     Serial_COM Inputs/GVL_Serial_Com.stComIn_SP1K2_PAX_PTM_01/D[9] <-> COM TxPDO-Map Inputs/Data In 9
//     Serial_COM Inputs/GVL_Serial_Com.stComIn_SP1K2_PAX_PTM_01/Status <-> COM TxPDO-Map Inputs/Status
//     Serial_COM Outputs/GVL_Serial_Com.stComOut_SP1K2_PAX_PTM_01/Ctrl <-> COM RxPDO-Map Outputs/Ctrl
//     Serial_COM Outputs/GVL_Serial_Com.stComOut_SP1K2_PAX_PTM_01/D[0] <-> COM RxPDO-Map Outputs/Data Out 0
//     Serial_COM Outputs/GVL_Serial_Com.stComOut_SP1K2_PAX_PTM_01/D[10] <-> COM RxPDO-Map Outputs/Data Out 10
//     Serial_COM Outputs/GVL_Serial_Com.stComOut_SP1K2_PAX_PTM_01/D[11] <-> COM RxPDO-Map Outputs/Data Out 11
//     Serial_COM Outputs/GVL_Serial_Com.stComOut_SP1K2_PAX_PTM_01/D[12] <-> COM RxPDO-Map Outputs/Data Out 12
//     Serial_COM Outputs/GVL_Serial_Com.stComOut_SP1K2_PAX_PTM_01/D[13] <-> COM RxPDO-Map Outputs/Data Out 13
//     Serial_COM Outputs/GVL_Serial_Com.stComOut_SP1K2_PAX_PTM_01/D[14] <-> COM RxPDO-Map Outputs/Data Out 14
//     Serial_COM Outputs/GVL_Serial_Com.stComOut_SP1K2_PAX_PTM_01/D[15] <-> COM RxPDO-Map Outputs/Data Out 15
//     Serial_COM Outputs/GVL_Serial_Com.stComOut_SP1K2_PAX_PTM_01/D[16] <-> COM RxPDO-Map Outputs/Data Out 16
//     Serial_COM Outputs/GVL_Serial_Com.stComOut_SP1K2_PAX_PTM_01/D[17] <-> COM RxPDO-Map Outputs/Data Out 17
//     Serial_COM Outputs/GVL_Serial_Com.stComOut_SP1K2_PAX_PTM_01/D[18] <-> COM RxPDO-Map Outputs/Data Out 18
//     Serial_COM Outputs/GVL_Serial_Com.stComOut_SP1K2_PAX_PTM_01/D[19] <-> COM RxPDO-Map Outputs/Data Out 19
//     Serial_COM Outputs/GVL_Serial_Com.stComOut_SP1K2_PAX_PTM_01/D[1] <-> COM RxPDO-Map Outputs/Data Out 1
//     Serial_COM Outputs/GVL_Serial_Com.stComOut_SP1K2_PAX_PTM_01/D[20] <-> COM RxPDO-Map Outputs/Data Out 20
//     Serial_COM Outputs/GVL_Serial_Com.stComOut_SP1K2_PAX_PTM_01/D[21] <-> COM RxPDO-Map Outputs/Data Out 21
//     Serial_COM Outputs/GVL_Serial_Com.stComOut_SP1K2_PAX_PTM_01/D[2] <-> COM RxPDO-Map Outputs/Data Out 2
//     Serial_COM Outputs/GVL_Serial_Com.stComOut_SP1K2_PAX_PTM_01/D[3] <-> COM RxPDO-Map Outputs/Data Out 3
//     Serial_COM Outputs/GVL_Serial_Com.stComOut_SP1K2_PAX_PTM_01/D[4] <-> COM RxPDO-Map Outputs/Data Out 4
//     Serial_COM Outputs/GVL_Serial_Com.stComOut_SP1K2_PAX_PTM_01/D[5] <-> COM RxPDO-Map Outputs/Data Out 5
//     Serial_COM Outputs/GVL_Serial_Com.stComOut_SP1K2_PAX_PTM_01/D[6] <-> COM RxPDO-Map Outputs/Data Out 6
//     Serial_COM Outputs/GVL_Serial_Com.stComOut_SP1K2_PAX_PTM_01/D[7] <-> COM RxPDO-Map Outputs/Data Out 7
//     Serial_COM Outputs/GVL_Serial_Com.stComOut_SP1K2_PAX_PTM_01/D[8] <-> COM RxPDO-Map Outputs/Data Out 8
//     Serial_COM Outputs/GVL_Serial_Com.stComOut_SP1K2_PAX_PTM_01/D[9] <-> COM RxPDO-Map Outputs/Data Out 9
//   plc_kfe_rix_vac Instance <-> Device 1 (EtherCAT)/Term 1 (EK1200)/Term 45 (EK1521-0010)/Term 47 (EK1501-0010)/Term 62 (EK1122)/Term 63 (EK1100) B950-233-100H1-R02-DRL-02/Term 98 (EK1122)/Term 156 (EK1100) B950-233-PAX-DRL-01/Term 163 (EL1004)
//     PlcTask Inputs/GVL_KFE_RIX_VAC.fb_SP1K2_PAX_PTM_02.i_xAtSpd <-> Channel 1/Input
//     PlcTask Inputs/GVL_KFE_RIX_VAC.fb_SP1K2_PAX_PTM_02.i_xFaultNC <-> Channel 3/Input
//     PlcTask Inputs/GVL_KFE_RIX_VAC.fb_SP1K2_PAX_PTM_02.i_xRemote <-> Channel 2/Input
//   plc_kfe_rix_vac Instance <-> Device 1 (EtherCAT)/Term 1 (EK1200)/Term 45 (EK1521-0010)/Term 47 (EK1501-0010)/Term 62 (EK1122)/Term 63 (EK1100) B950-233-100H1-R02-DRL-02/Term 98 (EK1122)/Term 156 (EK1100) B950-233-PAX-DRL-01/Term 165 (EL2004)
//     PlcTask Outputs/GVL_KFE_RIX_VAC.fb_SP1K2_PAX_PTM_02.q_PumpingStation <-> Channel 3/Output
//     PlcTask Outputs/GVL_KFE_RIX_VAC.fb_SP1K2_PAX_PTM_02.q_RunDO <-> Channel 1/Output
//     PlcTask Outputs/GVL_KFE_RIX_VAC.fb_SP1K2_PAX_PTM_02.q_xRemote <-> Channel 2/Output
//   plc_kfe_rix_vac Instance <-> Device 1 (EtherCAT)/Term 1 (EK1200)/Term 45 (EK1521-0010)/Term 47 (EK1501-0010)/Term 62 (EK1122)/Term 63 (EK1100) B950-233-100H1-R02-DRL-02/Term 98 (EK1122)/Term 156 (EK1100) B950-233-PAX-DRL-01/Term 166 (EL6021)
//     Serial_COM Inputs/GVL_Serial_Com.stComIn_SP1K2_PAX_PTM_02/D[0] <-> COM TxPDO-Map Inputs/Data In 0
//     Serial_COM Inputs/GVL_Serial_Com.stComIn_SP1K2_PAX_PTM_02/D[10] <-> COM TxPDO-Map Inputs/Data In 10
//     Serial_COM Inputs/GVL_Serial_Com.stComIn_SP1K2_PAX_PTM_02/D[11] <-> COM TxPDO-Map Inputs/Data In 11
//     Serial_COM Inputs/GVL_Serial_Com.stComIn_SP1K2_PAX_PTM_02/D[12] <-> COM TxPDO-Map Inputs/Data In 12
//     Serial_COM Inputs/GVL_Serial_Com.stComIn_SP1K2_PAX_PTM_02/D[13] <-> COM TxPDO-Map Inputs/Data In 13
//     Serial_COM Inputs/GVL_Serial_Com.stComIn_SP1K2_PAX_PTM_02/D[14] <-> COM TxPDO-Map Inputs/Data In 14
//     Serial_COM Inputs/GVL_Serial_Com.stComIn_SP1K2_PAX_PTM_02/D[15] <-> COM TxPDO-Map Inputs/Data In 15
//     Serial_COM Inputs/GVL_Serial_Com.stComIn_SP1K2_PAX_PTM_02/D[16] <-> COM TxPDO-Map Inputs/Data In 16
//     Serial_COM Inputs/GVL_Serial_Com.stComIn_SP1K2_PAX_PTM_02/D[17] <-> COM TxPDO-Map Inputs/Data In 17
//     Serial_COM Inputs/GVL_Serial_Com.stComIn_SP1K2_PAX_PTM_02/D[18] <-> COM TxPDO-Map Inputs/Data In 18
//     Serial_COM Inputs/GVL_Serial_Com.stComIn_SP1K2_PAX_PTM_02/D[19] <-> COM TxPDO-Map Inputs/Data In 19
//     Serial_COM Inputs/GVL_Serial_Com.stComIn_SP1K2_PAX_PTM_02/D[1] <-> COM TxPDO-Map Inputs/Data In 1
//     Serial_COM Inputs/GVL_Serial_Com.stComIn_SP1K2_PAX_PTM_02/D[20] <-> COM TxPDO-Map Inputs/Data In 20
//     Serial_COM Inputs/GVL_Serial_Com.stComIn_SP1K2_PAX_PTM_02/D[21] <-> COM TxPDO-Map Inputs/Data In 21
//     Serial_COM Inputs/GVL_Serial_Com.stComIn_SP1K2_PAX_PTM_02/D[2] <-> COM TxPDO-Map Inputs/Data In 2
//     Serial_COM Inputs/GVL_Serial_Com.stComIn_SP1K2_PAX_PTM_02/D[3] <-> COM TxPDO-Map Inputs/Data In 3
//     Serial_COM Inputs/GVL_Serial_Com.stComIn_SP1K2_PAX_PTM_02/D[4] <-> COM TxPDO-Map Inputs/Data In 4
//     Serial_COM Inputs/GVL_Serial_Com.stComIn_SP1K2_PAX_PTM_02/D[5] <-> COM TxPDO-Map Inputs/Data In 5
//     Serial_COM Inputs/GVL_Serial_Com.stComIn_SP1K2_PAX_PTM_02/D[6] <-> COM TxPDO-Map Inputs/Data In 6
//     Serial_COM Inputs/GVL_Serial_Com.stComIn_SP1K2_PAX_PTM_02/D[7] <-> COM TxPDO-Map Inputs/Data In 7
//     Serial_COM Inputs/GVL_Serial_Com.stComIn_SP1K2_PAX_PTM_02/D[8] <-> COM TxPDO-Map Inputs/Data In 8
//     Serial_COM Inputs/GVL_Serial_Com.stComIn_SP1K2_PAX_PTM_02/D[9] <-> COM TxPDO-Map Inputs/Data In 9
//     Serial_COM Inputs/GVL_Serial_Com.stComIn_SP1K2_PAX_PTM_02/Status <-> COM TxPDO-Map Inputs/Status
//     Serial_COM Outputs/GVL_Serial_Com.stComOut_SP1K2_PAX_PTM_02/Ctrl <-> COM RxPDO-Map Outputs/Ctrl
//     Serial_COM Outputs/GVL_Serial_Com.stComOut_SP1K2_PAX_PTM_02/D[0] <-> COM RxPDO-Map Outputs/Data Out 0
//     Serial_COM Outputs/GVL_Serial_Com.stComOut_SP1K2_PAX_PTM_02/D[10] <-> COM RxPDO-Map Outputs/Data Out 10
//     Serial_COM Outputs/GVL_Serial_Com.stComOut_SP1K2_PAX_PTM_02/D[11] <-> COM RxPDO-Map Outputs/Data Out 11
//     Serial_COM Outputs/GVL_Serial_Com.stComOut_SP1K2_PAX_PTM_02/D[12] <-> COM RxPDO-Map Outputs/Data Out 12
//     Serial_COM Outputs/GVL_Serial_Com.stComOut_SP1K2_PAX_PTM_02/D[13] <-> COM RxPDO-Map Outputs/Data Out 13
//     Serial_COM Outputs/GVL_Serial_Com.stComOut_SP1K2_PAX_PTM_02/D[14] <-> COM RxPDO-Map Outputs/Data Out 14
//     Serial_COM Outputs/GVL_Serial_Com.stComOut_SP1K2_PAX_PTM_02/D[15] <-> COM RxPDO-Map Outputs/Data Out 15
//     Serial_COM Outputs/GVL_Serial_Com.stComOut_SP1K2_PAX_PTM_02/D[16] <-> COM RxPDO-Map Outputs/Data Out 16
//     Serial_COM Outputs/GVL_Serial_Com.stComOut_SP1K2_PAX_PTM_02/D[17] <-> COM RxPDO-Map Outputs/Data Out 17
//     Serial_COM Outputs/GVL_Serial_Com.stComOut_SP1K2_PAX_PTM_02/D[18] <-> COM RxPDO-Map Outputs/Data Out 18
//     Serial_COM Outputs/GVL_Serial_Com.stComOut_SP1K2_PAX_PTM_02/D[19] <-> COM RxPDO-Map Outputs/Data Out 19
//     Serial_COM Outputs/GVL_Serial_Com.stComOut_SP1K2_PAX_PTM_02/D[1] <-> COM RxPDO-Map Outputs/Data Out 1
//     Serial_COM Outputs/GVL_Serial_Com.stComOut_SP1K2_PAX_PTM_02/D[20] <-> COM RxPDO-Map Outputs/Data Out 20
//     Serial_COM Outputs/GVL_Serial_Com.stComOut_SP1K2_PAX_PTM_02/D[21] <-> COM RxPDO-Map Outputs/Data Out 21
//     Serial_COM Outputs/GVL_Serial_Com.stComOut_SP1K2_PAX_PTM_02/D[2] <-> COM RxPDO-Map Outputs/Data Out 2
//     Serial_COM Outputs/GVL_Serial_Com.stComOut_SP1K2_PAX_PTM_02/D[3] <-> COM RxPDO-Map Outputs/Data Out 3
//     Serial_COM Outputs/GVL_Serial_Com.stComOut_SP1K2_PAX_PTM_02/D[4] <-> COM RxPDO-Map Outputs/Data Out 4
//     Serial_COM Outputs/GVL_Serial_Com.stComOut_SP1K2_PAX_PTM_02/D[5] <-> COM RxPDO-Map Outputs/Data Out 5
//     Serial_COM Outputs/GVL_Serial_Com.stComOut_SP1K2_PAX_PTM_02/D[6] <-> COM RxPDO-Map Outputs/Data Out 6
//     Serial_COM Outputs/GVL_Serial_Com.stComOut_SP1K2_PAX_PTM_02/D[7] <-> COM RxPDO-Map Outputs/Data Out 7
//     Serial_COM Outputs/GVL_Serial_Com.stComOut_SP1K2_PAX_PTM_02/D[8] <-> COM RxPDO-Map Outputs/Data Out 8
//     Serial_COM Outputs/GVL_Serial_Com.stComOut_SP1K2_PAX_PTM_02/D[9] <-> COM RxPDO-Map Outputs/Data Out 9
//   plc_kfe_rix_vac Instance <-> Device 1 (EtherCAT)/Term 1 (EK1200)/Term 45 (EK1521-0010)/Term 47 (EK1501-0010)/Term 62 (EK1122)/Term 63 (EK1100) B950-233-100H1-R02-DRL-02/Term 98 (EK1122)/Term 156 (EK1100) B950-233-PAX-DRL-01/Term 167 (EL2624)
//     PlcTask Outputs/GVL_KFE_RIX_VAC.fb_SP1K2_PAX_GCC_1.q_xHV_DIS <-> Channel 2/Output
//     PlcTask Outputs/GVL_KFE_RIX_VAC.fb_SP1K2_PAX_GCC_2.q_xHV_DIS <-> Channel 1/Output
//   plc_kfe_rix_vac Instance <-> Device 1 (EtherCAT)/Term 1 (EK1200)/Term 45 (EK1521-0010)/Term 47 (EK1501-0010)/Term 62 (EK1122)/Term 63 (EK1100) B950-233-100H1-R02-DRL-02/Term 98 (EK1122)/Term 156 (EK1100) B950-233-PAX-DRL-01/Term 168 (EL2004)
//     PlcTask Outputs/GVL_KFE_RIX_VAC.fb_SP1K2_PAX_VRC_4.q_xOPN_DO <-> Channel 1/Output
//   plc_kfe_rix_vac Instance <-> Device 1 (EtherCAT)/Term 1 (EK1200)/Term 45 (EK1521-0010)/Term 47 (EK1501-0010)/Term 62 (EK1122)/Term 63 (EK1100) B950-233-100H1-R02-DRL-02/Term 98 (EK1122)/Term 156 (EK1100) B950-233-PAX-DRL-01/Term 169 (EL1004)
//     PlcTask Inputs/GVL_KFE_RIX_VAC.fb_SP1K2_PAX_VRC_4.i_xClsLS <-> Channel 2/Input
//     PlcTask Inputs/GVL_KFE_RIX_VAC.fb_SP1K2_PAX_VRC_4.i_xOpnLS <-> Channel 1/Input
//   plc_kfe_rix_vac Instance <-> Device 1 (EtherCAT)/Term 1 (EK1200)/Term 45 (EK1521-0010)/Term 47 (EK1501-0010)/Term 62 (EK1122)/Term 63 (EK1100) B950-233-100H1-R02-DRL-02/Term 98 (EK1122)/Term 156 (EK1100) B950-233-PAX-DRL-01/Term 170 (EL3174-0002)
//     PlcTask Inputs/GVL_KFE_RIX_VAC.fb_SP1K2_PAX_GCC_1.i_iPRESS_R <-> AI Standard Channel 2/Value
//     PlcTask Inputs/GVL_KFE_RIX_VAC.fb_SP1K2_PAX_GCC_2.i_iPRESS_R <-> AI Standard Channel 4/Value
//     PlcTask Inputs/GVL_KFE_RIX_VAC.fb_SP1K2_PAX_GPI_1.i_iPRESS_R <-> AI Standard Channel 1/Value
//     PlcTask Inputs/GVL_KFE_RIX_VAC.fb_SP1K2_PAX_GPI_2.i_iPRESS_R <-> AI Standard Channel 3/Value
//   plc_kfe_rix_vac Instance <-> Device 1 (EtherCAT)/Term 1 (EK1200)/Term 45 (EK1521-0010)/Term 47 (EK1501-0010)/Term 62 (EK1122)/Term 63 (EK1100) B950-233-100H1-R02-DRL-02/Term 98 (EK1122)/Term 156 (EK1100) B950-233-PAX-DRL-01/Term 172 (EL1124)
//     PlcTask Inputs/GVL_KFE_RIX_VAC.fb_SP1K2_PAX_GCC_1.i_xDisc_Active <-> Channel 2/Input
//     PlcTask Inputs/GVL_KFE_RIX_VAC.fb_SP1K2_PAX_GCC_1.i_xHV_ON <-> Channel 1/Input
//   plc_kfe_rix_vac Instance <-> Device 1 (EtherCAT)/Term 1 (EK1200)/Term 45 (EK1521-0010)/Term 47 (EK1501-0010)/Term 91 (EL3174-0002)
//     PlcTask Inputs/GVL_KFE_RIX_VAC.fb_IM2K2_PPM_PIP_1.i_iPRESS <-> AI Standard Channel 1/GVL_KFE_RIX_VAC.fb_IM2K2_PPM_PIP_1.i_iPRESS
//     PlcTask Inputs/GVL_KFE_RIX_VAC.fb_IM3K2_PPM_PIP_1.i_iPRESS <-> AI Standard Channel 2/GVL_KFE_RIX_VAC.fb_IM3K2_PPM_PIP_1.i_iPRESS
//     PlcTask Inputs/GVL_KFE_RIX_VAC.fb_IM4K2_PPM_PIP_1.i_iPRESS <-> AI Standard Channel 3/GVL_KFE_RIX_VAC.fb_IM4K2_PPM_PIP_1.i_iPRESS
//     PlcTask Inputs/GVL_KFE_RIX_VAC.fb_LI2K2_K2A_PIP_1.i_iPRESS <-> AI Standard Channel 4/GVL_KFE_RIX_VAC.fb_LI2K2_K2A_PIP_1.i_iPRESS
//   plc_kfe_rix_vac Instance <-> Device 1 (EtherCAT)/Term 1 (EK1200)/Term 45 (EK1521-0010)/Term 47 (EK1501-0010)/Term 93 (EL1124)
//     PlcTask Inputs/GVL_KFE_RIX_VAC.fb_IM2K2_PPM_PIP_1.i_xError <-> Channel 2/GVL_KFE_RIX_VAC.fb_IM2K2_PPM_PIP_1.i_xError
//     PlcTask Inputs/GVL_KFE_RIX_VAC.fb_IM3K2_PPM_PIP_1.i_xError <-> Channel 4/GVL_KFE_RIX_VAC.fb_IM3K2_PPM_PIP_1.i_xError
//     PlcTask Inputs/GVL_KFE_RIX_VAC.fb_IM2K2_PPM_PIP_1.i_xIP_ON <-> Channel 1/GVL_KFE_RIX_VAC.fb_IM2K2_PPM_PIP_1.i_xIP_ON
//     PlcTask Inputs/GVL_KFE_RIX_VAC.fb_IM3K2_PPM_PIP_1.i_xIP_ON <-> Channel 3/GVL_KFE_RIX_VAC.fb_IM3K2_PPM_PIP_1.i_xIP_ON
//   plc_kfe_rix_vac Instance <-> Device 1 (EtherCAT)/Term 1 (EK1200)/Term 45 (EK1521-0010)/Term 47 (EK1501-0010)/Term 94 (EL1124)
//     PlcTask Inputs/GVL_KFE_RIX_VAC.fb_IM4K2_PPM_PIP_1.i_xError <-> Channel 2/GVL_KFE_RIX_VAC.fb_IM4K2_PPM_PIP_1.i_xError
//     PlcTask Inputs/GVL_KFE_RIX_VAC.fb_IM4K2_PPM_PIP_1.i_xIP_ON <-> Channel 1/GVL_KFE_RIX_VAC.fb_IM4K2_PPM_PIP_1.i_xIP_ON
//     PlcTask Inputs/GVL_KFE_RIX_VAC.fb_LI2K2_K2A_PIP_1.i_xError <-> Channel 4/GVL_KFE_RIX_VAC.fb_LI2K2_K2A_PIP_1.i_xError
//     PlcTask Inputs/GVL_KFE_RIX_VAC.fb_LI2K2_K2A_PIP_1.i_xIP_ON <-> Channel 3/GVL_KFE_RIX_VAC.fb_LI2K2_K2A_PIP_1.i_xIP_ON
//   plc_kfe_rix_vac Instance <-> Device 1 (EtherCAT)/Term 1 (EK1200)/Term 5 (EL1004)
//     PlcTask Inputs/GVL_KFE_RIX_VAC.fb_MR1K2_SWITCH_PIP_1.i_xSP_DI <-> Channel 3/Input
//     PlcTask Inputs/GVL_KFE_RIX_VAC.fb_PC1K1_ZOS_PIP_1.i_xSP_DI <-> Channel 2/Input
//     PlcTask Inputs/GVL_KFE_RIX_VAC.fb_TV1K1_PLEG_PIP_1.i_xSP_DI <-> Channel 4/Input
//   plc_kfe_rix_vac Instance <-> Device 1 (EtherCAT)/Term 1 (EK1200)/Term 6 (EL2794)
//     PlcTask Outputs/GVL_KFE_RIX_VAC.fb_SL1K2_EXIT_PIP_1.q_xHVEna_DO <-> Channel 1/Output
//   plc_kfe_rix_vac Instance <-> Device 1 (EtherCAT)/Term 1 (EK1200)/Term 7 (EL3064)
//     PlcTask Inputs/GVL_KFE_RIX_VAC.fb_SL1K2_EXIT_PIP_1.i_iPRESS <-> AI Standard Channel 1/Value
//   plc_kfe_rix_vac Instance <-> Device 1 (EtherCAT)/Term 1 (EK1200)/Term 8 (EL1004)
//     PlcTask Inputs/GVL_KFE_RIX_VAC.fb_SL1K2_EXIT_PIP_1.i_xSP_DI <-> Channel 1/Input
//   plc_kfe_rix_vac Instance <-> plc_kfe_rix_vac/plc_kfe_rix_vac Instance
//     FSTask Inputs/GVL_RIX_VAC_FS_DEVICES.fb_TV1K2_VFS_1.i_xCLS_SW <-> PlcTask Outputs/GVL_KFE_RIX_VAC.fb_TV1K2_VFS_Interface.q_xCLS_SW
//     FSTask Inputs/GVL_RIX_VAC_FS_DEVICES.fb_TV1K2_VFS_1.i_xOPN_SW <-> PlcTask Outputs/GVL_KFE_RIX_VAC.fb_TV1K2_VFS_Interface.q_xOPN_SW
//     FSTask Inputs/GVL_RIX_VAC_FS_DEVICES.fb_TV1K2_VFS_1.i_xOverrideMode <-> PlcTask Outputs/GVL_KFE_RIX_VAC.fb_TV1K2_VFS_Interface.q_xOverrideMode
//     FSTask Inputs/GVL_RIX_VAC_FS_DEVICES.fb_TV1K2_VFS_1.i_xOverrideOpen <-> PlcTask Outputs/GVL_KFE_RIX_VAC.fb_TV1K2_VFS_Interface.q_xOverrideOpen
//     FSTask Inputs/GVL_RIX_VAC_FS_DEVICES.fb_TV1K2_VFS_1.i_xPress_OK <-> PlcTask Outputs/GVL_KFE_RIX_VAC.fb_TV1K2_VFS_Interface.q_xPRESS_OK
//     FSTask Inputs/GVL_RIX_VAC_FS_DEVICES.fb_TV1K2_VFS_1.i_xVAC_FAULT_Reset <-> PlcTask Outputs/GVL_KFE_RIX_VAC.fb_TV1K2_VFS_Interface.q_xVAC_FAULT_Reset
//     FSTask Inputs/GVL_RIX_VAC_FS_DEVICES.fb_TV1K2_VFS_1.i_xVetoValveClosed <-> PlcTask Outputs/GVL_KFE_RIX_VAC.fb_TV1K2_VFS_Interface.q_xVetoValveClosed
//     FSTask Inputs/GVL_RIX_VAC_FS_DEVICES.fb_TV1K2_VFS_1.i_xVetoValveOpenDO <-> PlcTask Outputs/GVL_KFE_RIX_VAC.fb_TV1K2_VFS_Interface.q_xVetoValveOpenDO
//     FSTask Outputs/GVL_RIX_VAC_FS_DEVICES.fb_TV1K2_VFS_1.q_eVFS_State <-> PlcTask Inputs/GVL_KFE_RIX_VAC.fb_TV1K2_VFS_Interface.i_eVFS_State
//     FSTask Outputs/GVL_RIX_VAC_FS_DEVICES.fb_TV1K2_VFS_1.q_xMPS_OK <-> PlcTask Inputs/GVL_KFE_RIX_VAC.fb_TV1K2_VFS_Interface.i_xMPS_OK
//     FSTask Outputs/GVL_RIX_VAC_FS_DEVICES.fb_TV1K2_VFS_1.q_xTrigger <-> PlcTask Inputs/GVL_KFE_RIX_VAC.fb_TV1K2_VFS_Interface.i_xTrigger
//     FSTask Outputs/GVL_RIX_VAC_FS_DEVICES.fb_TV1K2_VFS_1.q_xVAC_FAULT_OK <-> PlcTask Inputs/GVL_KFE_RIX_VAC.fb_TV1K2_VFS_Interface.i_xVAC_FAULT_OK
//     FSTask Outputs/GVL_RIX_VAC_FS_DEVICES.fb_TV1K2_VFS_1.q_xVFS_Closed <-> PlcTask Inputs/GVL_KFE_RIX_VAC.fb_TV1K2_VFS_Interface.i_xVFS_Closed
//     FSTask Outputs/GVL_RIX_VAC_FS_DEVICES.fb_TV1K2_VFS_1.q_xVFS_Open <-> PlcTask Inputs/GVL_KFE_RIX_VAC.fb_TV1K2_VFS_Interface.i_xVFS_Open
//     PlcTask Inputs/GVL_KFE_RIX_VAC.fb_TV1K2_VFS_Interface.i_eVFS_State <-> FSTask Outputs/GVL_RIX_VAC_FS_DEVICES.fb_TV1K2_VFS_1.q_eVFS_State
//     PlcTask Inputs/GVL_KFE_RIX_VAC.fb_TV1K2_VFS_Interface.i_xMPS_OK <-> FSTask Outputs/GVL_RIX_VAC_FS_DEVICES.fb_TV1K2_VFS_1.q_xMPS_OK
//     PlcTask Inputs/GVL_KFE_RIX_VAC.fb_TV1K2_VFS_Interface.i_xTrigger <-> FSTask Outputs/GVL_RIX_VAC_FS_DEVICES.fb_TV1K2_VFS_1.q_xTrigger
//     PlcTask Inputs/GVL_KFE_RIX_VAC.fb_TV1K2_VFS_Interface.i_xVAC_FAULT_OK <-> FSTask Outputs/GVL_RIX_VAC_FS_DEVICES.fb_TV1K2_VFS_1.q_xVAC_FAULT_OK
//     PlcTask Inputs/GVL_KFE_RIX_VAC.fb_TV1K2_VFS_Interface.i_xVFS_Closed <-> FSTask Outputs/GVL_RIX_VAC_FS_DEVICES.fb_TV1K2_VFS_1.q_xVFS_Closed
//     PlcTask Inputs/GVL_KFE_RIX_VAC.fb_TV1K2_VFS_Interface.i_xVFS_Open <-> FSTask Outputs/GVL_RIX_VAC_FS_DEVICES.fb_TV1K2_VFS_1.q_xVFS_Open
//     PlcTask Outputs/GVL_KFE_RIX_VAC.fb_TV1K2_VFS_Interface.q_xCLS_SW <-> FSTask Inputs/GVL_RIX_VAC_FS_DEVICES.fb_TV1K2_VFS_1.i_xCLS_SW
//     PlcTask Outputs/GVL_KFE_RIX_VAC.fb_TV1K2_VFS_Interface.q_xOPN_SW <-> FSTask Inputs/GVL_RIX_VAC_FS_DEVICES.fb_TV1K2_VFS_1.i_xOPN_SW
//     PlcTask Outputs/GVL_KFE_RIX_VAC.fb_TV1K2_VFS_Interface.q_xOverrideMode <-> FSTask Inputs/GVL_RIX_VAC_FS_DEVICES.fb_TV1K2_VFS_1.i_xOverrideMode
//     PlcTask Outputs/GVL_KFE_RIX_VAC.fb_TV1K2_VFS_Interface.q_xOverrideOpen <-> FSTask Inputs/GVL_RIX_VAC_FS_DEVICES.fb_TV1K2_VFS_1.i_xOverrideOpen
//     PlcTask Outputs/GVL_KFE_RIX_VAC.fb_TV1K2_VFS_Interface.q_xPRESS_OK <-> FSTask Inputs/GVL_RIX_VAC_FS_DEVICES.fb_TV1K2_VFS_1.i_xPress_OK
//     PlcTask Outputs/GVL_KFE_RIX_VAC.fb_TV1K2_VFS_Interface.q_xVAC_FAULT_Reset <-> FSTask Inputs/GVL_RIX_VAC_FS_DEVICES.fb_TV1K2_VFS_1.i_xVAC_FAULT_Reset
//     PlcTask Outputs/GVL_KFE_RIX_VAC.fb_TV1K2_VFS_Interface.q_xVetoValveClosed <-> FSTask Inputs/GVL_RIX_VAC_FS_DEVICES.fb_TV1K2_VFS_1.i_xVetoValveClosed
//     PlcTask Outputs/GVL_KFE_RIX_VAC.fb_TV1K2_VFS_Interface.q_xVetoValveOpenDO <-> FSTask Inputs/GVL_RIX_VAC_FS_DEVICES.fb_TV1K2_VFS_1.i_xVetoValveOpenDO

// ---- GVLs/GVL_KFE_RIX_VAC.TcGVL
VAR_GLOBAL

// MKS275 Gauges

{attribute 'pytmc' := ' pv: PC1K1:ZOS:GPI:1 '}
fb_PC1K1_ZOS_GPI_1 : FB_MKS275;
{attribute 'pytmc' := ' pv: MR1K2:SWITCH:GPI:1 '}
fb_MR1K2_SWITCH_GPI_1 : FB_MKS275;
{attribute 'pytmc' := ' pv: TV1K1:PLEG:GPI:1 '}
fb_TV1K1_PLEG_GPI_1 : FB_MKS275;
{attribute 'TcLinkTo' := 	'.i_iPRESS_R	:= TIID^Device 1 (EtherCAT)^B950_100H1_WALL (EK1100)^Term 119 (EL3174)^AI Standard Channel 2^Value'}
{attribute 'pytmc' := ' pv: SL1K2:EXIT:GPI:1 '}
fb_SL1K2_EXIT_GPI_1 : FB_MKS275;
{attribute 'pytmc' := ' pv: MR2K2:FLAT:GPI:1 '}
fb_MR2K2_FLAT_GPI_1 : FB_MKS275;
{attribute 'pytmc' := ' pv: MR3K2:KBH:GPI:1 '}
fb_MR3K2_KBH_GPI_1 : FB_MKS275;
{attribute 'pytmc' := ' pv: MR4K2:KBV:GPI:1 '}
fb_MR4K2_KBV_GPI_1 : FB_MKS275;
{attribute 'TcLinkTo' := 	'.i_iPRESS_R	:= TIIB[Term 170 (EL3174-0002)]^AI Standard Channel 1^Value'}
{attribute 'pytmc' := ' pv: SP1K2:PAX:GPI:1 '}
fb_SP1K2_PAX_GPI_1 : FB_MKS275;
{attribute 'TcLinkTo' := 	'.i_iPRESS_R	:= TIIB[Term 170 (EL3174-0002)]^AI Standard Channel 3^Value'}
{attribute 'pytmc' := ' pv: SP1K2:PAX:GPI:2 '}
fb_SP1K2_PAX_GPI_2 : FB_MKS275;
{attribute 'TcLinkTo' := 	'.i_iPRESS_R	:= TIIB[EL3174_05_11]^AI Standard Channel 1^Value'}
{attribute 'pytmc' := ' pv: IM5K2:PPM:GPI:1 '}
fb_IM5K2_PPM_GPI_1 : FB_MKS275;


//New Superbee piranis
{attribute 'pytmc' := ' pv: TM2K2:ATM:GPI:1 '}
fb_TM2K2_ATM_GPI_1 : FB_MKS275;

{attribute 'TcLinkTo' := 	'.i_iPRESS_R	:= TIIB[Box 256 (EP3174-0002)]^AI Standard Channel 3^Value'}
{attribute 'pytmc' := ' pv: AT3K2:SOLID:GPI:1 '}
fb_AT3K2_SOLID_GPI_1 : FB_MKS275;


//MKS275 EP Gauges
{attribute 'TcLinkTo' := 	'.i_iPRESS_R	:= TIID^Device 1 (EtherCAT)^Term 1 (EK1200)^Term 45 (EK1521-0010)^Term 47 (EK1501-0010)^Term 62 (EK1122)^Box 111 (EP3174-0002)^AI Standard Channel 2^Value'}
{attribute 'pytmc' := ' pv: ST1K2:PPS:GPI:1 '}
fb_ST1K2_PPS_GPI_1 : FB_MKS275;

// MKS500 Gauges

{attribute 'pytmc' := ' pv: PC1K1:ZOS:GCC:1 '}
fb_PC1K1_ZOS_GCC_1 : FB_MKS500;
{attribute 'pytmc' := ' pv: MR1K2:SWITCH:GCC:1 '}
fb_MR1K2_SWITCH_GCC_1 : FB_MKS500;
{attribute 'pytmc' := ' pv: TV1K1:PLEG:GCC:1 '}
fb_TV1K1_PLEG_GCC_1 : FB_MKS500;

{attribute 'TcLinkTo' := 	'.i_iPRESS_R	:=	TIID^Device 1 (EtherCAT)^B950_100H1_WALL (EK1100)^Term 119 (EL3174)^AI Standard Channel 1^Value;
                                 .i_xHV_ON	    :=	TIID^Device 1 (EtherCAT)^B950_100H1_WALL (EK1100)^Term 123 (EL1124)^Channel 1^Input;
                                 .i_xDisc_Active:=	TIID^Device 1 (EtherCAT)^B950_100H1_WALL (EK1100)^Term 123 (EL1124)^Channel 2^Input;
                                 .q_xHV_DIS		:= 	TIID^Device 1 (EtherCAT)^B950_100H1_WALL (EK1100)^Term 118 (EL2624)^Channel 1^Output	'}
{attribute 'pytmc' := ' pv: SL1K2:EXIT:GCC:1 '}
fb_SL1K2_EXIT_GCC_1 : FB_MKS500;
{attribute 'pytmc' := ' pv: MR2K2:FLAT:GCC:1 '}
fb_MR2K2_FLAT_GCC_1 : FB_MKS500;
{attribute 'pytmc' := ' pv: IM2K2:PPM:GCC:1 '}
fb_IM2K2_PPM_GCC_1 : FB_MKS500;
{attribute 'pytmc' := ' pv: MR3K2:KBH:GCC:1 '}
fb_MR3K2_KBH_GCC_1 : FB_MKS500;
{attribute 'pytmc' := ' pv: IM3K2:PPM:GCC:1 '}
fb_IM3K2_PPM_GCC_1 : FB_MKS500;
{attribute 'pytmc' := ' pv: MR4K2:KBV:GCC:1 '}
fb_MR4K2_KBV_GCC_1 : FB_MKS500;
{attribute 'pytmc' := ' pv: IM4K2:PPM:GCC:1 '}
fb_IM4K2_PPM_GCC_1 : FB_MKS500;
{attribute 'pytmc' := ' pv: IM5K2:PPM:GCC:1 '}
fb_IM5K2_PPM_GCC_1 : FB_MKS500;
{attribute 'pytmc' := ' pv: TM2K2:K2B:GCC:1 '}
fb_TM2K2_K2B_GCC_1 : FB_MKS500;
{attribute 'TcLinkTo' := 	'.i_iPRESS_R	:=	TIIB[Term 170 (EL3174-0002)]^AI Standard Channel 2^Value;
                                 .i_xHV_ON	    :=	TIIB[Term 172 (EL1124)]^Channel 1^Input;
                                 .i_xDisc_Active:=	TIIB[Term 172 (EL1124)]^Channel 2^Input;
                                 .q_xHV_DIS		:= 	TIIB[Term 167 (EL2624)]^Channel 2^Output'}
{attribute 'pytmc' := ' pv: SP1K2:PAX:GCC:1 '}
fb_SP1K2_PAX_GCC_1 : FB_MKS500;

//New Televac gauge
{attribute 'TcLinkTo' := 	'.i_iPRESS_R	:=	TIIB[Term 170 (EL3174-0002)]^AI Standard Channel 4^Value;
                              .q_xHV_DIS		:= 	TIIB[Term 167 (EL2624)]^Channel 1^Output'}
{attribute 'pytmc' := ' pv: SP1K2:PAX:GCC:2 '}
fb_SP1K2_PAX_GCC_2 : FB_MX7M;

//MKS500 EP Gauges
{attribute 'TcLinkTo' := 	'.i_iPRESS_R	:=	TIID^Device 1 (EtherCAT)^Term 1 (EK1200)^Term 45 (EK1521-0010)^Term 47 (EK1501-0010)^Term 62 (EK1122)^Box 111 (EP3174-0002)^AI Standard Channel 1^Value;
                             .q_xHV_DIS		:= 	TIID^Device 1 (EtherCAT)^Term 1 (EK1200)^Term 45 (EK1521-0010)^Term 47 (EK1501-0010)^Term 62 (EK1122)^K2S2-DRL-01 (EP2624-0002)^Channel 1^Output	'}
{attribute 'pytmc' := ' pv: ST1K2:PPS:GCC:1 '}
fb_ST1K2_PPS_GCC_1 : FB_MKS500;


//MKS972B Combo Gauges

{attribute 'TcLinkTo' := 	'.i_iPRESS_R	:=	TIIB[Box 256 (EP3174-0002)]^AI Standard Channel 2^Value'}
{attribute 'pytmc' := ' pv: AT3K2:SOLID:GCP:1 '}
fb_AT3K2_SOLID_GCP_1 : FB_972;

{attribute 'TcLinkTo' := 	'.i_iPRESS_R	:=	TIIB[Box 256 (EP3174-0002)]^AI Standard Channel 4^Value'}
{attribute 'pytmc' :=' pv: SP2K2:TXAS:GCP:1 '}
fb_SP2K2_TXAS_GCP_1 : FB_972;


// MKS422
{attribute 'pytmc' := ' pv: TV4K2:GFS:1 '}
fb_TV4K2_GFS_1 : FB_MKS422;


// VGC Valves

{attribute 'pytmc' := ' pv: MR1K2:SWITCH:VGC:1 '}
fb_MR1K2_SWITCH_VGC_1 : FB_VGC;
{attribute 'pytmc' := ' pv: MR1K2:SWITCH:VGC:2 '}
fb_MR1K2_SWITCH_VGC_2 : FB_VGC;

{attribute 'TcLinkTo' := 	'.i_xOpnLS	:=	TIID^Device 1 (EtherCAT)^B950_100H1_WALL (EK1100)^Term 120 (EL1004)^Channel 1^Input;
                                 .i_xClsLS	:=	TIID^Device 1 (EtherCAT)^B950_100H1_WALL (EK1100)^Term 120 (EL1004)^Channel 2^Input;
                                .q_xOPN_DO	:=	TIID^Device 1 (EtherCAT)^B950_100H1_WALL (EK1100)^Term 121 (EL2004)^Channel 1^Output'}
{attribute 'pytmc' := ' pv: SL1K2:EXIT:VGC:1 '}
fb_SL1K2_EXIT_VGC_1 : FB_VGC;
{attribute 'pytmc' := ' pv: MR2K2:FLAT:VGC:1 '}
fb_MR2K2_FLAT_VGC_1 : FB_VGC;
{attribute 'pytmc' := ' pv: MR2K2:FLAT:VGC:2 '}
fb_MR2K2_FLAT_VGC_2 : FB_VGC;
{attribute 'pytmc' := ' pv: MR3K2:KBH:VGC:1 '}
fb_MR3K2_KBH_VGC_1 : FB_VGC;
{attribute 'pytmc' := ' pv: MR3K2:KBH:VGC:2 '}
fb_MR3K2_KBH_VGC_2 : FB_VGC;
{attribute 'pytmc' := ' pv: MR4K2:KBV:VGC:1 '}
fb_MR4K2_KBV_VGC_1 : FB_VGC;
{attribute 'pytmc' := ' pv: MR4K2:KBV:VGC:2 '}
fb_MR4K2_KBV_VGC_2 : FB_VGC;
{attribute 'pytmc' := ' pv: LI3K2:K2B:VWC:1 '}
fb_LI3K2_K2B_VWC_1 : FB_VGC;
{attribute 'TcLinkTo' := 	'.i_xOpnLS		 :=	TIIB[EL1004_05_01]^Channel 3^Input;
                                 .i_xClsLS	 := TIIB[EL1004_05_01]^Channel 4^Input ;
                                 .q_xOPN_DO  := TIIB[EL2004_05_02]^Channel 2^Output'}
{attribute 'pytmc' := ' pv: LI2K2:K2A:VWC:1 '}
fb_LI2K2_K2A_VWC_1 : FB_VGC;

// VGC EP Valves
{attribute 'TcLinkTo' := 	'.i_xOpnLS	:=	TIID^Device 1 (EtherCAT)^Term 1 (EK1200)^Term 45 (EK1521-0010)^Term 47 (EK1501-0010)^Term 62 (EK1122)^Box 110 (EP2338-0002)^Channel 1^Input;
                                 .i_xClsLS	:=	TIID^Device 1 (EtherCAT)^Term 1 (EK1200)^Term 45 (EK1521-0010)^Term 47 (EK1501-0010)^Term 62 (EK1122)^Box 110 (EP2338-0002)^Channel 2^Input;
                                .q_xOPN_DO	:=	TIID^Device 1 (EtherCAT)^Term 1 (EK1200)^Term 45 (EK1521-0010)^Term 47 (EK1501-0010)^Term 62 (EK1122)^Box 110 (EP2338-0002)^Channel 11^Output'}
{attribute 'pytmc' := ' pv: ST1K2:PPS:VGC:1 '}
fb_ST1K2_PPS_VGC_1 : FB_VGC;
{attribute 'TcLinkTo' := 	'.i_xOpnLS	:=	TIID^Device 1 (EtherCAT)^Term 1 (EK1200)^Term 45 (EK1521-0010)^Term 47 (EK1501-0010)^Term 62 (EK1122)^Box 110 (EP2338-0002)^Channel 5^Input;
                                 .i_xClsLS	:=	TIID^Device 1 (EtherCAT)^Term 1 (EK1200)^Term 45 (EK1521-0010)^Term 47 (EK1501-0010)^Term 62 (EK1122)^Box 110 (EP2338-0002)^Channel 6^Input;
                                .q_xOPN_DO	:=	TIID^Device 1 (EtherCAT)^Term 1 (EK1200)^Term 45 (EK1521-0010)^Term 47 (EK1501-0010)^Term 62 (EK1122)^Box 110 (EP2338-0002)^Channel 15^Output'}
{attribute 'pytmc' := ' pv: SP1K2:PAX:VGC:1 '}
fb_SP1K2_PAX_VGC_1 : FB_VGC;


//SP1K2 VRCs
{attribute 'pytmc' := ' pv: SP1K2:PAX:VRC:1 '}
{attribute 'TcLinkTo' := 	'.i_xOpnLS		 :=	TIIB[Term 157 (EL1004)]^Channel 1^Input;
                                 .i_xClsLS	 := TIIB[Term 157 (EL1004)]^Channel 2^Input ;
                                 .q_xOPN_DO  := TIIB[Term 158 (EL2004)]^Channel 1^Output'}
fb_SP1K2_PAX_VRC_1 : FB_VRC;
{attribute 'pytmc' := ' pv: SP1K2:PAX:VRC:2 '}
{attribute 'TcLinkTo' := 	'.i_xOpnLS		:=	TIIB[Term 157 (EL1004)]^Channel 3^Input;
                                 .i_xClsLS		:= TIIB[Term 157 (EL1004)]^Channel 4^Input ;
                                 .q_xOPN_DO	:= TIIB[Term 158 (EL2004)]^Channel 2^Output'}
fb_SP1K2_PAX_VRC_2 : FB_VRC;
{attribute 'pytmc' := ' pv: SP1K2:PAX:VRM:3 '}
{attribute 'TcLinkTo' := 	'.i_xOpnLS		:=	TIIB[Term 159 (EL1004)]^Channel 1^Input;
                                 .i_xClsLS		:= TIIB[Term 159 (EL1004)]^Channel 2^Input ;
                                 .q_xOPN_DO	:= TIIB[Term 158 (EL2004)]^Channel 3^Output'}
fb_SP1K2_PAX_VRM_3 : FB_VRC;
{attribute 'pytmc' := ' pv: SP1K2:PAX:VRC:4 '}
{attribute 'TcLinkTo' := 	'.i_xOpnLS		:=	TIIB[Term 169 (EL1004)]^Channel 1^Input;
                                 .i_xClsLS		:= TIIB[Term 169 (EL1004)]^Channel 2^Input ;
                                 .q_xOPN_DO	:= TIIB[Term 168 (EL2004)]^Channel 1^Output'}
fb_SP1K2_PAX_VRC_4 : FB_VRC;

{attribute 'pytmc' := ' pv: AT3K2:SOLID:VWC:01'}
{attribute 'TcLinkTo' := 	'.i_xOpnLS		:=	TIIB[K2S18_EL1004_E1]^Channel 1^Input;
                             .i_xClsLS		:= TIIB[K2S18_EL1004_E1]^Channel 2^Input ;
                             .q_xCLS_DO	:= TIIB[K2S18_EL2004_E2]^Channel 1^Output'}
fb_AT3K2_SOLID_VWC_01 : FB_VRC_NO_FFO;

//{attribute 'pytmc' := ' pv: SP1K2:PAX:VRC:5 '}
//{attribute 'TcLinkTo' := 	'.i_xOpnLS		:=	TIIB[Term 169 (EL1004)]^Channel 3^Input;
//                                .i_xClsLS		:= TIIB[Term 169 (EL1004)]^Channel 4^Input ;
//                                 .q_xOPN_DO	:= TIIB[Term 168 (EL2004)]^Channel 2^Output'}
//fb_SP1K2_PAX_VRC_5 : FB_VRC; (Not beign installed currently)

// PIP_Gamma Pumps

{attribute 'pytmc' := ' pv: PC1K1:ZOS:PIP:1 '}
fb_PC1K1_ZOS_PIP_1 : FB_PIP_GAMMA;
//{attribute 'pytmc' := ' pv: PC1K1:ZOS:PIP:2 '}
//fb_PC1K1_ZOS_PIP_2 : FB_PIP_GAMMA;
{attribute 'pytmc' := ' pv: MR1K2:SWITCH:PIP:1 '}
fb_MR1K2_SWITCH_PIP_1 : FB_PIP_GAMMA;
{attribute 'pytmc' := ' pv: TV1K1:PLEG:PIP:1 '}
fb_TV1K1_PLEG_PIP_1 : FB_PIP_GAMMA;
{attribute 'TcLinkTo' := 	'.i_iPRESS		:=	TIIB[B950_233_R02 (E3) (EL3064)]^AI Standard Channel 1^GVL_KFE_RIX_VAC.fb_ST1K2_PPS_PIP_1.i_iPRESS;
                                 .i_xSP_DI		:=  TIIB[B950_233_R02 (E4) (EL1004)]^Channel 1^GVL_KFE_RIX_VAC.fb_ST1K2_PPS_PIP_1.i_xSP_DI;
                                 .q_xHVEna_DO	:= TIIB[B950_233_R02 (E2) (EL2794)]^Channel 1^GVL_KFE_RIX_VAC.fb_ST1K2_PPS_PIP_1.q_xHVEna_DO'}
{attribute 'pytmc' := ' pv: ST1K2:PPS:PIP:1 '}
fb_ST1K2_PPS_PIP_1 : FB_PIP_GAMMA;

{attribute 'TcLinkTo' := 	'.i_iPRESS		:=	TIIB[Term 7 (EL3064)]^AI Standard Channel 1^Value;
                                 .i_xSP_DI		:=  TIIB[Term 8 (EL1004)]^Channel 1^Input;
                                 .q_xHVEna_DO	:= TIIB[Term 6 (EL2794)]^Channel 1^Output'}
{attribute 'pytmc' := ' pv: SL1K2:EXIT:PIP:1 '}
fb_SL1K2_EXIT_PIP_1 : FB_PIP_GAMMA;
{attribute 'pytmc' := ' pv: MR2K2:FLAT:PIP:1 '}
fb_MR2K2_FLAT_PIP_1 : FB_PIP_GAMMA;
{attribute 'pytmc' := ' pv: MR3K2:KBH:PIP:1 '}
fb_MR3K2_KBH_PIP_1 : FB_PIP_GAMMA;
{attribute 'pytmc' := ' pv: MR4K2:KBV:PIP:1 '}
fb_MR4K2_KBV_PIP_1 : FB_PIP_GAMMA;
{attribute 'pytmc' := ' pv: TV4K2:PIP:1 '}
fb_TV4K2_PIP_1 : FB_PIP_GAMMA;
{attribute 'pytmc' := ' pv: IM5K2:PPM:PIP:1 '}
fb_IM5K2_PPM_PIP_1 : FB_PIP_GAMMA;
{attribute 'pytmc' := ' pv: PA1K2:PIP:1 '}
fb_PA1K2_PIP_1 : FB_PIP_GAMMA;

{attribute 'pytmc' := ' pv: SP1K2:PAX:PIP:1 '}
{attribute 'TcLinkTo' := 	'.i_iPRESS		:= TIID^Device 1 (EtherCAT)^Term 1 (EK1200)^Term 45 (EK1521-0010)^Term 47 (EK1501-0010)^Term 53 (EL3064)^AI Standard Channel 2^Value ;
                               .q_xHVEna_DO 	:= TIID^Device 1 (EtherCAT)^Term 1 (EK1200)^Term 45 (EK1521-0010)^Term 47 (EK1501-0010)^Term 52 (EL2794)^Channel 2^Output ;
                               .i_xSP_DI		:= TIID^Device 1 (EtherCAT)^Term 1 (EK1200)^Term 45 (EK1521-0010)^Term 47 (EK1501-0010)^Term 54 (EL1004)^Channel 2^Input '}
fb_SP1K2_PAX_PIP_1 : FB_PIP_GAMMA;

//SIP PIP NexTORR Pumps
{attribute 'pytmc' := ' pv: IM2K2:PPM:PIP:1 '}
fb_IM2K2_PPM_PIP_1 : FB_PIP_SIP;
{attribute 'pytmc' := ' pv: IM3K2:PPM:PIP:1 '}
fb_IM3K2_PPM_PIP_1 : FB_PIP_SIP;
{attribute 'pytmc' := ' pv: IM4K2:PPM:PIP:1 '}
fb_IM4K2_PPM_PIP_1 : FB_PIP_SIP;
{attribute 'pytmc' := ' pv: LI2K2:K2A:PIP:1 '}
fb_LI2K2_K2A_PIP_1 : FB_PIP_SIP;
{attribute 'pytmc' := ' pv: SP2K2:TXAS:PIP:1 '}
fb_SP2K2_TXAS_PIP_1 : FB_PIP_SIP;


//PAX Turbo pumps (Pfeiffer turbo pumps TC400 *)

{attribute 'pytmc' := ' pv: SP1K2:PAX:PTM:1 '}
{attribute 'TcLinkTo' := 	'.i_xAtSpd		      := TIIB[Term 160 (EL1004)]^Channel 1^Input ;
                               .i_xRemote 	      := TIIB[Term 160 (EL1004)]^Channel 2^Input ;
                               .i_xFaultNC		  := TIIB[Term 160 (EL1004)]^Channel 3^Input;
                               .q_RunDO           := TIIB[Term 161 (EL2004)]^Channel 1^Output;
                               .q_xRemote         := TIIB[Term 161 (EL2004)]^Channel 2^Output ;
                               .q_PumpingStation  := TIIB[Term 161 (EL2004)]^Channel 3^Output'}
fb_SP1K2_PAX_PTM_01 : FB_PTM_Pfeiffer;
{attribute 'pytmc' := ' pv: SP1K2:PAX:PTM:2 '}
{attribute 'TcLinkTo' := 	'.i_xAtSpd		      := TIIB[Term 163 (EL1004)]^Channel 1^Input ;
                               .i_xRemote 	      := TIIB[Term 163 (EL1004)]^Channel 2^Input ;
                               .i_xFaultNC		  := TIIB[Term 163 (EL1004)]^Channel 3^Input;
                               .q_RunDO           := TIIB[Term 165 (EL2004)]^Channel 1^Output;
                               .q_xRemote         := TIIB[Term 165 (EL2004)]^Channel 2^Output ;
                               .q_PumpingStation  := TIIB[Term 165 (EL2004)]^Channel 3^Output'}
fb_SP1K2_PAX_PTM_02 : FB_PTM_Pfeiffer;

{attribute 'pytmc' := ' pv: LI3K2:K2B_OUT:PTM:01 '}
{attribute 'TcLinkTo' := 	'.i_xAtSpd		      := TIIB[EL1004_05_03]^Channel 1^Input ;
                               .i_xRemote 	      := TIIB[EL1004_05_03]^Channel 2^Input ;
                               .i_xFaultNC		  := TIIB[EL1004_05_03]^Channel 3^Input;
                               .q_RunDO           := TIIB[EL2004_05_04]^Channel 1^Output;
                               .q_xRemote         := TIIB[EL2004_05_04]^Channel 2^Output ;
                               .q_PumpingStation  := TIIB[EL2004_05_04]^Channel 3^Output'}
fb_LI3K2_K2B_OUT_PTM_01 : FB_PTM_Pfeiffer;


{attribute 'pytmc' := ' pv: LI4K2:K2B_OUT:PTM:01 '}
{attribute 'TcLinkTo' := 	'.i_xAtSpd		      := TIIB[K2S18 _EL1004_E4]^Channel 1^Input ;
                               .i_xRemote 	      := TIIB[K2S18 _EL1004_E4]^Channel 2^Input ;
                               .i_xFaultNC		  := TIIB[K2S18 _EL1004_E4]^Channel 3^Input;
                               .q_RunDO           := TIIB[K2S18_EL2004_E5]^Channel 1^Output;
                               .q_xRemote         := TIIB[K2S18_EL2004_E5]^Channel 2^Output ;
                               .q_PumpingStation  := TIIB[K2S18_EL2004_E5]^Channel 3^Output'}
fb_LI4K2_K2B_OUT_PTM_01 : FB_PTM_Pfeiffer;


//VFS

{attribute 'pytmc' := '		pv: TV1K2:VFS:1	'}
    {attribute 'TcLinkTo' := 	'.q_xPress_OK		:= 	TIPC^plc_kfe_rix_vac^plc_kfe_rix_vac Instance^FSTask Inputs^GVL_RIX_VAC_FS_DEVICES.fb_TV1K2_VFS_1.i_xPress_OK;
                                    .q_xOPN_SW			:=  TIPC^plc_kfe_rix_vac^plc_kfe_rix_vac Instance^FSTask Inputs^GVL_RIX_VAC_FS_DEVICES.fb_TV1K2_VFS_1.i_xOPN_SW;
                               .q_xCLS_SW			:=  TIPC^plc_kfe_rix_vac^plc_kfe_rix_vac Instance^FSTask Inputs^GVL_RIX_VAC_FS_DEVICES.fb_TV1K2_VFS_1.i_xCLS_SW;
                             .q_xVAC_FAULT_Reset:= 	TIPC^plc_kfe_rix_vac^plc_kfe_rix_vac Instance^FSTask Inputs^GVL_RIX_VAC_FS_DEVICES.fb_TV1K2_VFS_1.i_xVAC_FAULT_Reset;
                             .q_xOverrideMode	:= 	TIPC^plc_kfe_rix_vac^plc_kfe_rix_vac Instance^FSTask Inputs^GVL_RIX_VAC_FS_DEVICES.fb_TV1K2_VFS_1.i_xOverrideMode;
                                 .q_xOverrideOpen	:= TIPC^plc_kfe_rix_vac^plc_kfe_rix_vac Instance^FSTask Inputs^GVL_RIX_VAC_FS_DEVICES.fb_TV1K2_VFS_1.i_xOverrideOpen;
                                 .i_xTrigger		:=	TIPC^plc_kfe_rix_vac^plc_kfe_rix_vac Instance^FSTask Outputs^GVL_RIX_VAC_FS_DEVICES.fb_TV1K2_VFS_1.q_xTrigger;
                                 .i_xVFS_Open		:= TIPC^plc_kfe_rix_vac^plc_kfe_rix_vac Instance^FSTask Outputs^GVL_RIX_VAC_FS_DEVICES.fb_TV1K2_VFS_1.q_xVFS_Open;
                                 .i_xVFS_Closed		:=	TIPC^plc_kfe_rix_vac^plc_kfe_rix_vac Instance^FSTask Outputs^GVL_RIX_VAC_FS_DEVICES.fb_TV1K2_VFS_1.q_xVFS_Closed;
                             .i_xVAC_FAULT_OK	:=  TIPC^plc_kfe_rix_vac^plc_kfe_rix_vac Instance^FSTask Outputs^GVL_RIX_VAC_FS_DEVICES.fb_TV1K2_VFS_1.q_xVAC_FAULT_OK;
                             .i_xMPS_OK			:=  TIPC^plc_kfe_rix_vac^plc_kfe_rix_vac Instance^FSTask Outputs^GVL_RIX_VAC_FS_DEVICES.fb_TV1K2_VFS_1.q_xMPS_OK;
                             .i_eVFS_State		:=	TIPC^plc_kfe_rix_vac^plc_kfe_rix_vac Instance^FSTask Outputs^GVL_RIX_VAC_FS_DEVICES.fb_TV1K2_VFS_1.q_eVFS_State;
                                 .q_xVetoValveOpenDO := TIPC^plc_kfe_rix_vac^plc_kfe_rix_vac Instance^FSTask Inputs^GVL_RIX_VAC_FS_DEVICES.fb_TV1K2_VFS_1.i_xVetoValveOpenDO;
                                 .q_xVetoValveClosed := TIPC^plc_kfe_rix_vac^plc_kfe_rix_vac Instance^FSTask Inputs^GVL_RIX_VAC_FS_DEVICES.fb_TV1K2_VFS_1.i_xVetoValveClosed	'}
fb_TV1K2_VFS_Interface : FB_VFS_Interface;


//Interface for KFE Valve - SP1K1-MONO-VGC-2
{attribute 'pytmc' :=' pv: PC1K1:ZOS:GCC:1:ILK'}
    st_RIX_ILK			:	ST_EXT_ILK;

    {attribute 'TcLinkTo' := 	'.q_xILK_OK_DO	:= TIID^Device 1 (EtherCAT)^Term 1 (EK1200)^Term 11 (EL2794)^Channel 1^Output '}

    fb_RIX_ILK			:	FB_EXT_ILK;


(*Pfeiffer serial*)
stPfeiffer_CTRL_SP1K2_PAX_PTM_01     : ARRAY[1..gcMaxPfeifferPumps] OF ST_PfeifferControl;
stPfeiffer_RBK_SP1K2_PAX_PTM_01      : ARRAY[1..gcMaxPfeifferPumps] OF ST_PfeifferStatus;
fbPfeifferCom_SP1K2_PAX_PTM_01       : FB_PFEIFFER_COM;

stPfeiffer_CTRL_SP1K2_PAX_PTM_02     : ARRAY[1..gcMaxPfeifferPumps] OF ST_PfeifferControl;
stPfeiffer_RBK_SP1K2_PAX_PTM_02      : ARRAY[1..gcMaxPfeifferPumps] OF ST_PfeifferStatus;
fbPfeifferCom_SP1K2_PAX_PTM_02       : FB_PFEIFFER_COM;

stPfeiffer_CTRL_LI3K2_PAX_PTM_01    : ARRAY[1..gcMaxPfeifferPumps] OF ST_PfeifferControl;
stPfeiffer_RBK_LI3K2_PAX_PTM_01      : ARRAY[1..gcMaxPfeifferPumps] OF ST_PfeifferStatus;
fbPfeifferCom_LI3K2_PAX_PTM_01       : FB_PFEIFFER_COM;

stPfeiffer_CTRL_LI4K2_PAX_PTM_01     : ARRAY[1..gcMaxPfeifferPumps] OF ST_PfeifferControl;
stPfeiffer_RBK_LI4K2_PAX_PTM_01      : ARRAY[1..gcMaxPfeifferPumps] OF ST_PfeifferStatus;
fbPfeifferCom_LI4K2_PAX_PTM_01       : FB_PFEIFFER_COM;


//// Connected to B950-310-WALL-W-DRL-02 (Mechanical Room )
{attribute 'pytmc' := ' pv: RIXS:PRO:01 '}
{attribute 'TcLinkTo' := '.q_xMPStart := TIIB[EL2794_03_03]^Channel 1^Output;
                          .q_xBPStart := TIIB[EL2794_03_03]^Channel 2^Output;
                          .i_xMPStatus := TIIB[EL1088_03_01]^Channel 1^Input;
                          .i_xBPStatus := TIIB[EL1088_03_01]^Channel 2^Input;
                          .i_xWarning := TIIB[EL1088_03_01]^Channel 3^Input;
                          .i_xAlarmOK := TIIB[EL1088_03_01]^Channel 4^Input;
                          .i_xRemote := TIIB (EL1088_03_01]^Channel 5^Input
'}
RIXS_PRO_01 : FB_EbaraDryPump;
{attribute 'pytmc' := ' pv: RIXS:ROUGH:GPI:01 '}
{attribute 'TcLinkTo' := 	'.i_iPRESS_R	:=	TIIB[EL3174-0002_03_07]^AI Standard Channel 4^Value'}
RIXS_ROUGH_GPI_01 : FB_MKS275;

//VRO
{attribute 'pytmc' := ' pv: RIXS:ROUGH:VRO:01 '}
{attribute 'TcLinkTo' := 	'.q_xOPN_DO	:=	TIIB[EL2212_03_04]^DOX Control Channel 1^Control^Output'}
RIXS_ROUGH_VRO_01 : FB_VVC;

// IM6K2 PUMP

{attribute 'pytmc' := ' pv: IM6K2:TXAS:PTM:01 '}
{attribute 'TcLinkTo' := 	'.i_xAtSpd		      := TIIB[K2S18_EL1004_E7]^Channel 1^Input ;
                               .i_xRemote 	      := TIIB[K2S18_EL1004_E7]^Channel 2^Input ;
                               .i_xFaultNC		  := TIIB[K2S18_EL1004_E7]^Channel 3^Input;
                               .q_RunDO           := TIIB[K2S18_EL2004_E8]^Channel 1^Output;
                               .q_xRemote         := TIIB[K2S18_EL2004_E8]^Channel 2^Output ;
                               .q_PumpingStation  := TIIB[K2S18_EL2004_E8]^Channel 3^Output'}
fb_IM6K2_TXAS_PTM_01 : FB_PTM_Pfeiffer;

stPfeiffer_CTRL_IM6K2_TXAS_PTM_01     : ARRAY[1..gcMaxPfeifferPumps] OF ST_PfeifferControl;
stPfeiffer_RBK_IM6K2_TXAS_PTM_01      : ARRAY[1..gcMaxPfeifferPumps] OF ST_PfeifferStatus;
fbPfeifferCom_IM6K2_TXAS_PTM_01       : FB_PFEIFFER_COM;

END_VAR

// ---- GVLs/GVL_Serial_Com.TcGVL
//{attribute 'qualified_only'}
VAR_GLOBAL
    //COMM FUNCTION
    SerialRXBuffer_SP1K2_PAX_PTM_01     : ComBuffer;
    SerialTXBuffer_SP1K2_PAX_PTM_01     : ComBuffer;
    SerialRXBuffer_SP1K2_PAX_PTM_02     : ComBuffer;
    SerialTXBuffer_SP1K2_PAX_PTM_02     : ComBuffer;

    SerialRXBuffer_LI3K2_K2B_OUT_PTM_01     : ComBuffer;
     SerialTXBuffer_LI3K2_K2B_OUT_PTM_01     : ComBuffer;
    SerialRXBuffer_LI4K2_K2B_OUT_PTM_01     : ComBuffer;
     SerialTXBuffer_LI4K2_K2B_OUT_PTM_01     : ComBuffer;

    SerialRXBuffer_IM6K2_TXAS_PTM_01     : ComBuffer;
    SerialTXBuffer_IM6K2_TXAS_PTM_01     : ComBuffer;


    //Serial Terminal
    fbSerialLineControl_SP1K2_PAX_PTM_01     : SerialLineControl;
    fbSerialLineControl_SP1K2_PAX_PTM_02     : SerialLineControl;

    fbSerialLineControl_LI3K2_K2B_OUT_PTM_01     : SerialLineControl;
    fbSerialLineControl_LI4K2_K2B_OUT_PTM_01     : SerialLineControl;

    fbSerialLineControl_IM6K2_TXAS_PTM_01     : SerialLineControl;


    //SERIAL IO
    {attribute	'TcLinkTo'	:=	'.Status:=TIIB[Term 162 (EL6021)]^COM TxPDO-Map Inputs^Status;
                                 .D[0]:=TIIB[Term 162 (EL6021)]^COM TxPDO-Map Inputs^Data In 0;
                                 .D[1]:=TIIB[Term 162 (EL6021)]^COM TxPDO-Map Inputs^Data In 1;
                                 .D[2]:=TIIB[Term 162 (EL6021)]^COM TxPDO-Map Inputs^Data In 2;
                                 .D[3]:=TIIB[Term 162 (EL6021)]^COM TxPDO-Map Inputs^Data In 3;
                                 .D[4]:=TIIB[Term 162 (EL6021)]^COM TxPDO-Map Inputs^Data In 4;
                                 .D[5]:=TIIB[Term 162 (EL6021)]^COM TxPDO-Map Inputs^Data In 5;
                                 .D[6]:=TIIB[Term 162 (EL6021)]^COM TxPDO-Map Inputs^Data In 6;
                                 .D[7]:=TIIB[Term 162 (EL6021)]^COM TxPDO-Map Inputs^Data In 7;
                                 .D[8]:=TIIB[Term 162 (EL6021)]^COM TxPDO-Map Inputs^Data In 8;
                                 .D[9]:=TIIB[Term 162 (EL6021)]^COM TxPDO-Map Inputs^Data In 9;
                                 .D[10]:=TIIB[Term 162 (EL6021)]^COM TxPDO-Map Inputs^Data In 10;
                                 .D[11]:=TIIB[Term 162 (EL6021)]^COM TxPDO-Map Inputs^Data In 11;
                                 .D[12]:=TIIB[Term 162 (EL6021)]^COM TxPDO-Map Inputs^Data In 12;
                                 .D[13]:=TIIB[Term 162 (EL6021)]^COM TxPDO-Map Inputs^Data In 13;
                                 .D[14]:=TIIB[Term 162 (EL6021)]^COM TxPDO-Map Inputs^Data In 14;
                                 .D[15]:=TIIB[Term 162 (EL6021)]^COM TxPDO-Map Inputs^Data In 15;
                                 .D[16]:=TIIB[Term 162 (EL6021)]^COM TxPDO-Map Inputs^Data In 16;
                                 .D[17]:=TIIB[Term 162 (EL6021)]^COM TxPDO-Map Inputs^Data In 17;
                                 .D[18]:=TIIB[Term 162 (EL6021)]^COM TxPDO-Map Inputs^Data In 18;
                                 .D[19]:=TIIB[Term 162 (EL6021)]^COM TxPDO-Map Inputs^Data In 19;
                                 .D[20]:=TIIB[Term 162 (EL6021)]^COM TxPDO-Map Inputs^Data In 20;
                                 .D[21]:=TIIB[Term 162 (EL6021)]^COM TxPDO-Map Inputs^Data In 21
    '}
    stComIn_SP1K2_PAX_PTM_01 AT %I* : EL6inData22B;

    {attribute 'TcLinkTo'	:=	'.Ctrl:=TIIB[Term 162 (EL6021)]^COM RxPDO-Map Outputs^Ctrl;
                                 .D[0]:=TIIB[Term 162 (EL6021)]^COM RxPDO-Map Outputs^Data Out 0;
                                 .D[1]:=TIIB[Term 162 (EL6021)]^COM RxPDO-Map Outputs^Data Out 1;
                                 .D[2]:=TIIB[Term 162 (EL6021)]^COM RxPDO-Map Outputs^Data Out 2;
                                 .D[3]:=TIIB[Term 162 (EL6021)]^COM RxPDO-Map Outputs^Data Out 3;
                                 .D[4]:=TIIB[Term 162 (EL6021)]^COM RxPDO-Map Outputs^Data Out 4;
                                 .D[5]:=TIIB[Term 162 (EL6021)]^COM RxPDO-Map Outputs^Data Out 5;
                                 .D[6]:=TIIB[Term 162 (EL6021)]^COM RxPDO-Map Outputs^Data Out 6;
                                 .D[7]:=TIIB[Term 162 (EL6021)]^COM RxPDO-Map Outputs^Data Out 7;
                                 .D[8]:=TIIB[Term 162 (EL6021)]^COM RxPDO-Map Outputs^Data Out 8;
                                 .D[9]:=TIIB[Term 162 (EL6021)]^COM RxPDO-Map Outputs^Data Out 9;
                                 .D[10]:=TIIB[Term 162 (EL6021)]^COM RxPDO-Map Outputs^Data Out 10;
                                 .D[11]:=TIIB[Term 162 (EL6021)]^COM RxPDO-Map Outputs^Data Out 11;
                                 .D[12]:=TIIB[Term 162 (EL6021)]^COM RxPDO-Map Outputs^Data Out 12;
                                 .D[13]:=TIIB[Term 162 (EL6021)]^COM RxPDO-Map Outputs^Data Out 13;
                                 .D[14]:=TIIB[Term 162 (EL6021)]^COM RxPDO-Map Outputs^Data Out 14;
                                 .D[15]:=TIIB[Term 162 (EL6021)]^COM RxPDO-Map Outputs^Data Out 15;
                                 .D[16]:=TIIB[Term 162 (EL6021)]^COM RxPDO-Map Outputs^Data Out 16;
                                 .D[17]:=TIIB[Term 162 (EL6021)]^COM RxPDO-Map Outputs^Data Out 17;
                                 .D[18]:=TIIB[Term 162 (EL6021)]^COM RxPDO-Map Outputs^Data Out 18;
                                 .D[19]:=TIIB[Term 162 (EL6021)]^COM RxPDO-Map Outputs^Data Out 19;
                                 .D[20]:=TIIB[Term 162 (EL6021)]^COM RxPDO-Map Outputs^Data Out 20;
                                 .D[21]:=TIIB[Term 162 (EL6021)]^COM RxPDO-Map Outputs^Data Out 21
    '}
    stComOut_SP1K2_PAX_PTM_01 AT %Q* : EL6outData22B;

